//############################################################################
// Local time; used for timestamps
//############################################################################
GVL_MSG_XTS.fbLocalTime();
GVL_MSG_XTS.sLocalTime                              := GVL_MSG_XTS.fbLocalTime.LocalTimeString;
GVL_MSG_XTS.dtLocalTime                             := GVL_MSG_XTS.fbLocalTime.LocalTime;
//############################################################################
//############################################################################
// 	example for init sequence
//############################################################################	
CASE eInit
OF
  E_PROGRESS.PROGRESS_INVALID:
    // In the beginning there was no error...
    eInitError                                  := E_PROGRESS.PROGRESS_NOT_EXIST;
    //---------------------------------------------------------------------------
    // where are the stations?
    // TODO: after importing this project into your XTS TwinCAT solution
    //       setup of Station parameters is required.
    //---------------------------------------------------------------------------
    // default initialization, please leave this in here
    DefaultStationParameters();        
    //---------------------------------------------------------------------------
    //---------------------------------------------------------------------------
    // where to start?
    // fb_TransportUnit is connected StationStartIndex and StationStart
    //
    // TODO: after importing this project into your XTS TwinCAT solution
    //       setup of StartStation parameters is up to you to decide.
    //---------------------------------------------------------------------------
    GVL_XTS.StationStartIndex                   := 1; // this index is yours to change, fbTransportUnit is connected to it
    GVL_XTS.StationStart                        := GVL_XTS.StationParameter[GVL_XTS.StationStartIndex]; // put in here any plausible data you like
    //---------------------------------------------------------------------------

    eInit                                       := E_PROGRESS.PROGRESS_BUSY;
    // clear command interface
    GVL_XTS.XpuCtrl.Cmd                         := E_XPU_CTRL.XTS_CMD_NULL;
    GVL_MSG_XTS.TransportMessageCtrl.Cmd            := E_MESSAGE_CTRL.MSG_CTRL_NULL;
    GVL_MSG_XTS.MetricsMessageCtrl.Cmd              := E_MESSAGE_CTRL.MSG_CTRL_NULL;

    // set detailed message levvel for startup
    GVL_MSG_XTS.MessageLevelXpu                     := E_MessageType.eMessageVerbose; //GVL_MSG.MessageLevel;
    GVL_XTS.CaGroup.MessageLevel                := E_MessageType.eMessageVerbose; //GVL_MSG.MessageLevel;
    GVL_XTS.XtsTransport.MessageLevel           := E_MessageType.eMessageVerbose; //GVL_MSG.MessageLevel;

    FOR nStation := 1 TO MAX_STATION
    DO
      GVL_MSG_XTS.MessageLevelStations[nStation]    := E_MessageType.eMessageVerbose; //GVL_MSG.MessageLevel;
    END_FOR
    FOR nMover := 1 TO MAX_MOVER
    DO
      GVL_MSG_XTS.MessageLevelMovers[nMover]        := E_MessageType.eMessageVerbose; //GVL_MSG.MessageLevel;
    END_FOR
    
  //-----------------------------------------------------------------------------
  //-----------------------------------------------------------------------------
  E_PROGRESS.PROGRESS_BUSY:         // init Xpu, ProcessingUnit, MotorModules
    eInit                                       := E_PROGRESS.PROGRESS_PREPARE;
    GVL_MSG_XTS.TransportMessageCtrl.Cmd            := E_MESSAGE_CTRL.MSG_CTRL_INIT;
    GVL_MSG_XTS.MetricsMessageCtrl.Cmd              := E_MESSAGE_CTRL.MSG_CTRL_INIT;


  //-----------------------------------------------------------------------------
  //-----------------------------------------------------------------------------
  E_PROGRESS.PROGRESS_PREPARE:      // wait for init to be done
    GVL_XTS.XpuCtrl.Cmd                         := E_XPU_CTRL.XTS_CMD_INIT;
    IF (GVL_XTS.XpuState.State      = E_XPU_STATE.XTS_INIT + E_PROGRESS.PROGRESS_ERROR)
    THEN
      stMsg.eType                               := E_MessageType.eMessageInfo;
      stMsg.eDevice                             := e_Device.Device_Main;
      stMsg.eSubdevice                          := e_Subdevice.MainInit;
      stMsg.iErrorNumber                        := GVL_XTS.XpuState.Check;
      stMsg.sText                               := concat('MAIN.eInit Error: ', TO_STRING(MAIN_XTS.eInit));
      stMsg.sText                               := concat(stMsg.sText , ': ');
      stMsg.sText                               := concat(stMsg.sText, 'XpuState.Check: ');
      stMsg.sText                               := concat(stMsg.sText, TO_STRING(GVL_XTS.XpuState.Check));
      f_MessageSet(stMsg);

      eInitError                                := eInit;
      eInit                                     := E_PROGRESS.PROGRESS_ERROR;

    ELSIF (GVL_XTS.XpuState.State   = E_XPU_STATE.XTS_INIT + E_PROGRESS.PROGRESS_DONE)
    THEN
      eInit                                     := E_PROGRESS.PROGRESS_STARTUP;
      GVL_XTS.XpuCtrl.Cmd                       := E_XPU_CTRL.XTS_IDLE;
    END_IF

  //-----------------------------------------------------------------------------
  //-----------------------------------------------------------------------------
  E_PROGRESS.PROGRESS_STARTUP:
    CASE GVL_XTS.XpuState.Check
    OF
      E_XPU_CHECK.MOVER_ID_SIMULATION,
      E_XPU_CHECK.MOVER_ID_DETECTION_VALID:
        IF (GVL_XTS.XpuState.State = E_XPU_STATE.XTS_IDLE + E_PROGRESS.PROGRESS_WORKING)
        THEN
          eInit                                     := E_PROGRESS.PROGRESS_CHECK;
        END_IF
    END_CASE
  //-----------------------------------------------------------------------------
  //-----------------------------------------------------------------------------
  E_PROGRESS.PROGRESS_CHECK:
    eInit                                       := E_PROGRESS.PROGRESS_OCCUPIED;

    FOR nStation := 1 TO MAX_STATION
    DO
      GVL_MSG_XTS.MessageLevelStations[nStation]    := GVL_MSG_XTS.MessageLevel;
    END_FOR
    FOR nMover := 1 TO MAX_MOVER
    DO
      GVL_MSG_XTS.MessageLevelMovers[nMover]        := GVL_MSG_XTS.MessageLevel;
    END_FOR

  //-----------------------------------------------------------------------------
  //-----------------------------------------------------------------------------
  E_PROGRESS.PROGRESS_OCCUPIED:
    //---------------------------------------------------------------------------
    // how many nests to start with?
    // - this is for you to decide and me to secure, 
    //    so leave the initialisation as it is
    //
    // TODO: after importing this project into your XTS TwinCAT solution
    //       setup of StartStation NestMask configuration is up to you to decide.
    //---------------------------------------------------------------------------
    IF (GVL_XTS.XtsTransport.StationStartIndex > 0) AND
       (GVL_XTS.XtsTransport.StationStartIndex < MAX_STATION+1)
    THEN
      GVL_XTS.StationStart.nConfiguredStopCount := GVL_XTS.StationParameter[GVL_XTS.XtsTransport.StationStartIndex].nConfiguredStopCount;
    END_IF
    eInit                                       := E_PROGRESS.PROGRESS_WORKING;

  //-----------------------------------------------------------------------------
  //-----------------------------------------------------------------------------
  E_PROGRESS.PROGRESS_WORKING:
    GVL_MSG_XTS.TransportMessageCtrl.Cmd            := E_MESSAGE_CTRL.MSG_CTRL_WRITE;
    eInit                                       := E_PROGRESS.PROGRESS_DONE;

    stMsg.eType                                 := E_MessageType.eMessageInfo;
    stMsg.eDevice                               := e_Device.Device_Main;
    stMsg.eSubdevice                            := e_Subdevice.MainInit;
    stMsg.iErrorNumber                          := GVL_XTS.XpuState.Check;
    stMsg.sText                                 := concat('MAIN.eInit Done: ', TO_STRING(MAIN_XTS.eInit));
    stMsg.sText                                 := concat(stMsg.sText , ': ');
    stMsg.sText                                 := concat(stMsg.sText, 'XpuState.Check: ');
    stMsg.sText                                 := concat(stMsg.sText, TO_STRING(GVL_XTS.XpuState.Check));
    f_MessageSet(stMsg);

    //---------------------------------------------------------------------------
END_CASE
//############################################################################
//############################################################################
// 	/XTS Transport Unit
//############################################################################
//  - main control function block for transport layer
//  - requires access to member controls
//    - Xpu
//    - CaGroup
//    - Mover
//    - Station Control
//    - Station LinkedList Interface
//############################################################################
//
// cyclic call
GVL_XTS.XtsTransport();

// main control
GVL_XTS.XtsTransport.Ctrl                       REF= GVL_XTS.XtsTransportCtrl;   // main control
GVL_XTS.XtsTransport.State                      REF= GVL_XTS.XtsTransportState;  // main state
                                        
// member controls                      
GVL_XTS.XtsTransport.XpuCtrl                    REF= GVL_XTS.XpuCtrl;
GVL_XTS.XtsTransport.XpuState                   REF= GVL_XTS.XpuState;
GVL_XTS.XtsTransport.XpuInfo                    REF= GVL_XTS.XpuInfo;
                                        
GVL_XTS.XtsTransport.GroupItf                   :=   GVL_XTS.CaGroupItf;
GVL_XTS.XtsTransport.GroupInfo                  REF= GVL_XTS.CaGroupInfo;
                                        
GVL_XTS.XtsTransport.MoverItf                   REF= GVL_XTS.MoverItf;
GVL_XTS.XtsTransport.MoverInfo                  REF= GVL_XTS.MoverInfo;
GVL_XTS.XtsTransport.MoverLastPosition          REF= GVL_XTS.LastPosition;
GVL_XTS.XtsTransport.MoverLastGap               REF= GVL_XTS.LastGap;

GVL_XTS.XtsTransport.StationStartIndex          :=   GVL_XTS.StationStartIndex;                                        
GVL_XTS.XtsTransport.StationStart               REF= GVL_XTS.StationStart;      // start position for E_XTS_TRANSPORT_CTRL.CMD_TRANSPORT_START
GVL_XTS.XtsTransport.StationCtrlItf             REF= GVL_XTS.StationCtrlItf;    // station interfaces are required for accessing station methods
GVL_XTS.XtsTransport.StationListsItf            REF= GVL_XTS.StationListItf;    // list interface is required for access to linked list methods
GVL_XTS.XtsTransport.StationControl             REF= GVL_XTS.StationCtrl;
GVL_XTS.XtsTransport.StationState               REF= GVL_XTS.StationState;
//############################################################################
// 	XTS Transport Unit/
//############################################################################
//############################################################################
//############################################################################
// 	/XTS Stations
//############################################################################	
FOR nStation := 1 TO MAX_STATION
DO
  // epimetheus assembles the body
  GVL_XTS.StationListItf[nStation]              := GVL_XTS.StationList[nStation];   // interfaces for list methods
  GVL_XTS.StationCtrlItf[nStation]              := GVL_XTS.Station[nStation];       // interfaces for station methods

  CASE GVL_XTS.StationParameter[nStation].eType
  OF
    //-----------------------------------------------------------------------------
    E_STATION_TYPE.STATION_PROCESS:
      GVL_XTS.Station[nStation].MessageLevel    := GVL_MSG_XTS.MessageLevelStations[nStation];

      GVL_XTS.Station[nStation].StationId       := nStation;  // Know Thyself!

    
      GVL_XTS.Station[nStation].Ctrl            REF= GVL_XTS.StationCtrl;           // station ctrl from extern
      GVL_XTS.Station[nStation].State           REF= GVL_XTS.StationState;          // station state to extern
    
      GVL_XTS.Station[nStation].ItfStations     REF= GVL_XTS.StationListItf;        // give every station all list interfaces for writing mover tickets
      GVL_XTS.Station[nStation].ItfMover        REF= GVL_XTS.MoverItf;              // give every station all mover interfaces for movement in / out of station
      GVL_XTS.Station[nStation].Mover           REF= GVL_XTS.AxisRefMover;          // AXIS_REF to read infos from
      GVL_XTS.Station[nStation].MoverOffset     REF= GVL_XTS.PositionOffset;        // static offsets for all stations, all movers, all stop positions
    
      GVL_XTS.Station[nStation].StationParameter  REF= GVL_XTS.StationParameter;// give every station all station parameters for sending to WaitPos of target station
    
      // cyclic call
      GVL_XTS.Station[nStation].Cycle();                                        // cycle for handshaking with extern
    
      // Queue data for each station
      GVL_XTS.StationQueue[nStation]            := GVL_XTS.StationListItf[nStation].Data;


    //-----------------------------------------------------------------------------
    E_STATION_TYPE.STATION_GEAR_IN_POS:
      GVL_XTS.StationGearIn[nStation].MessageLevel:= GVL_MSG_XTS.MessageLevelStations[nStation];

      GVL_XTS.StationGearIn[nStation].StationId   := nStation;  // Know Thyself!
    
      GVL_XTS.StationGearIn[nStation].Ctrl        REF= GVL_XTS.StationCtrl;           // station ctrl from extern
      GVL_XTS.StationGearIn[nStation].State       REF= GVL_XTS.StationState;          // station state to extern
    
      GVL_XTS.StationGearIn[nStation].ItfStations REF= GVL_XTS.StationListItf;        // give every station all list interfaces for writing mover tickets
      GVL_XTS.StationGearIn[nStation].ItfMover    REF= GVL_XTS.MoverItf;              // give every station all mover interfaces for movement in / out of station
      GVL_XTS.StationGearIn[nStation].Mover       REF= GVL_XTS.AxisRefMover;          // AXIS_REF to read infos from
      GVL_XTS.StationGearIn[nStation].MoverOffset REF= GVL_XTS.PositionOffset;        // static offsets for all stations, all movers, all stop positions
    
    
      GVL_XTS.StationGearIn[nStation].StationParameter  REF= GVL_XTS.StationParameter;// give every station all station parameters for sending to WaitPos of target station
    
      // cyclic call
      GVL_XTS.StationGearIn[nStation].Cycle();                                        // cycle for handshaking with extern
    
      // Queue data for each station
      GVL_XTS.StationQueue[nStation]            := GVL_XTS.StationListItf[nStation].Data;
  ELSE
      //---------------------------------------------------------------------------------
      // no valid station type --> no identity
      //---------------------------------------------------------------------------------
      GVL_XTS.Station[nStation].StationId       := 0; // I am no one
      //---------------------------------------------------------------------------------
  END_CASE
END_FOR
//############################################################################
// 	XTS Stations/
//############################################################################	
//############################################################################
//############################################################################
// 	/XPU environment
//############################################################################	
GVL_XTS.Xpu.XpuInstance                         :=   1;
GVL_XTS.Xpu.MessageLevel                        :=   GVL_MSG_XTS.MessageLevelXpu;

GVL_XTS.Xpu.Ctrl                                REF= GVL_XTS.XpuCtrl;
GVL_XTS.Xpu.State                               REF= GVL_XTS.XpuState;
GVL_XTS.Xpu.XpuModuleInfoData                   REF= GVL_XTS.XpuModules;

GVL_XTS.Xpu.CaGroupOID                          :=   GVL_XTS.CaGroup.GroupInfo.CaGroupOID;

// cyclic call                                
GVL_XTS.Xpu();                                
GVL_XTS.XpuInfo                                 :=   GVL_XTS.Xpu.XpuInfo;
//############################################################################
// 	XPU environment/
//############################################################################	
//############################################################################
//############################################################################	
// 	/CA-Group Class
//############################################################################
// message device identifier
GVL_XTS.CaGroup.MessageDeviceIndex              :=   e_Device.CaGroup + 1;	
// assignment
GVL_XTS.CaGroup.AxisRef                         REF= GVL_XTS.AxisRefMover;
// Interface to Mover methods
GVL_XTS.CaGroup.MoverItf                        REF= GVL_XTS.MoverItf; 
GVL_XTS.CaGroup.GroupRef                        REF= GVL_XTS.CaGroupRef;
GVL_XTS.CaGroup.XpuInfo                         REF= GVL_XTS.XpuInfo;
// cyclic call
GVL_XTS.CaGroup.InfoCycle(TRUE);                // read group status
// InfoData from group
GVL_XTS.CaGroupInfo                             :=   GVL_XTS.CaGroup.GroupInfo;
// Interface of CaGroup
GVL_XTS.CaGroupItf                              :=   GVL_XTS.CaGroup;
//############################################################################	
// 	CA-Group Class/
//############################################################################
//############################################################################
//############################################################################
//  /Mover Class	
//############################################################################	
FOR nMover := 1 TO MAX_MOVER
DO
  GVL_XTS.Mover[nMover].MoverId                 :=   nMover;
  GVL_XTS.Mover[nMover].RailLength              :=   GVL_XTS.Xpu.RailLength;  // mover needs RailLength, in order to calc absolute position from modulo input
  GVL_XTS.Mover[nMover].MessageLevel            :=   GVL_MSG_XTS.MessageLevelMovers[nMover];

  GVL_XTS.Mover[nMover].Ctrl                    REF= GVL_XTS.MoverCtrl;       // mover control from extern
  GVL_XTS.Mover[nMover].State                   REF= GVL_XTS.MoverState;      // mover state to extern

  GVL_XTS.Mover[nMover].MoveData                REF= GVL_XTS.MoveData;        // dyn constraints for extern to write
  GVL_XTS.Mover[nMover].GearData                REF= GVL_XTS.GearData;        // GearIn/GearInPosCa data fro extern to write

  // assignment
  GVL_XTS.Mover[nMover].Mover                   REF= GVL_XTS.AxisRefMover[nMover];  // axis reference to Mover function block
  GVL_XTS.Mover[nMover].LastGap                 REF= GVL_XTS.LastGap[nMover];       // reference to last used gap value datafield
  GVL_XTS.Mover[nMover].LastPosition            REF= GVL_XTS.LastPosition[nMover];  // reference to last position datafield

  GVL_XTS.Mover[nMover].MoverInfo		            REF= GVL_XTS.MoverInfo[nMover];     // refernence to mover info data (ActPos, SetPos, ...)

  GVL_XTS.MoverItf[nMover]                      :=   GVL_XTS.Mover[nMover];

  // cyclic call
  GVL_XTS.Mover[nMover].Cycle();                // call AXIS_REF()
  GVL_XTS.Mover[nMover]();                      // call Ctrl/State
END_FOR
//############################################################################
//  Mover Class/	
//############################################################################	
//############################################################################
//############################################################################
//  /Mover Selector	
//############################################################################
GVL_XTS.MoverSelector.Ctrl                      REF= GVL_XTS.MoverSelectorCtrl;
GVL_XTS.MoverSelector.State                     REF= GVL_XTS.MoverSelectorState;
GVL_XTS.MoverSelector.AxisRef                   REF= GVL_XTS.AxisRefMover;
GVL_XTS.MoverSelector.Info                      REF= GVL_XTS.MoverInfo;
GVL_XTS.MoverSelector.ItfMover                  REF= GVL_XTS.MoverItf;

GVL_XTS.MoverSelector();
//############################################################################
//  Mover Selector/	
//############################################################################	
//############################################################################
//############################################################################
//  /logging
//    - all life is problem solving
//############################################################################
GVL_MSG_XTS.TransportMessageData.Ctrl               REF= GVL_MSG_XTS.TransportMessageCtrl;
GVL_MSG_XTS.TransportMessageData.State              REF= GVL_MSG_XTS.TransportMessageState;
GVL_MSG_XTS.TransportMessageData.MessageIndex       REF= GVL_MSG_XTS.MessageTransportIndex;
GVL_MSG_XTS.TransportMessageData.ErrorIndex         REF= GVL_MSG_XTS.MessageTransportError;
GVL_MSG_XTS.TransportMessageData.DirRoot            :=   ADR(GVL_MSG_XTS.LOG_DIR);
GVL_MSG_XTS.TransportMessageData.FileRoot           :=   ADR(GVL_MSG_XTS.LOG_FILE);
GVL_MSG_XTS.TransportMessageData.MsgList            :=   ADR(GVL_MSG_XTS.TransportMessages);
GVL_MSG_XTS.TransportMessageData.LocalTime          :=   ADR(GVL_MSG_XTS.dtLocalTime);
GVL_MSG_XTS.TransportMessageData();
eMsgState                                       :=   f_GetState   (GVL_MSG_XTS.TransportMessageState.State);
eMsgProgress                                    :=   f_GetProgress(GVL_MSG_XTS.TransportMessageState.State);

CASE eMsgState
OF
  E_MESSAGE_STATE.MSG_STATE_NULL:
    CASE eMsgProgress
    OF
      E_PROGRESS.PROGRESS_INVALID,
      E_PROGRESS.PROGRESS_DONE:
        IF (GVL_MSG_XTS.MessageTransportIndex > GVL_MSG_XTS.MAX_MESSAGE/100) OR
           (GVL_MSG_XTS.MessageTransportError > 0)
        THEN
          GVL_MSG_XTS.TransportMessageCtrl.Cmd      := E_MESSAGE_CTRL.MSG_CTRL_WRITE;
        ELSE
          tonIdleWriteMotion(IN := TRUE, PT:= tIdleWriteMotion);
          IF (tonIdleWriteMotion.Q)
          THEN
            GVL_MSG_XTS.TransportMessageCtrl.Cmd    := E_MESSAGE_CTRL.MSG_CTRL_WRITE;
          END_IF
        END_IF
    END_CASE

  E_MESSAGE_STATE.MSG_STATE_WRITE:
    CASE eMsgProgress
    OF
      E_PROGRESS.PROGRESS_ERROR,
      E_PROGRESS.PROGRESS_DONE:
          tonIdleWriteMotion(IN := FALSE, PT:= tIdleWriteMotion);
        GVL_MSG_XTS.TransportMessageCtrl.Cmd        := E_MESSAGE_CTRL.MSG_CTRL_NULL;
    END_CASE

ELSE
    CASE eMsgProgress
    OF
      E_PROGRESS.PROGRESS_DONE:
        GVL_MSG_XTS.TransportMessageCtrl.Cmd        := E_MESSAGE_CTRL.MSG_CTRL_NULL;
    END_CASE
END_CASE
//############################################################################
//  logging/
//############################################################################
//############################################################################
//############################################################################
//  /Transport Metrics
//############################################################################
GVL_MSG_XTS.MetricsMessageData.Ctrl                 REF= GVL_MSG_XTS.MetricsMessageCtrl;
GVL_MSG_XTS.MetricsMessageData.State                REF= GVL_MSG_XTS.MetricsMessageState;

GVL_MSG_XTS.MetricsMessageData.MessageIndex         REF= GVL_MSG_XTS.MessageMetricsIndex;
GVL_MSG_XTS.MetricsMessageData.ErrorIndex           REF= GVL_MSG_XTS.MessageMetricsError;

GVL_MSG_XTS.MetricsMessageData.DirRoot              :=   ADR(GVL_MSG_XTS.LOG_DIR);
GVL_MSG_XTS.MetricsMessageData.FileRoot             :=   ADR(GVL_MSG_XTS.LOG_FILE_METRIC);

GVL_MSG_XTS.MetricsMessageData.MsgList              :=   ADR(GVL_MSG_XTS.MetricsMessages);
GVL_MSG_XTS.MetricsMessageData.LocalTime            :=   ADR(GVL_MSG_XTS.dtLocalTime);

GVL_MSG_XTS.MetricsMessageData();

eMtrState                                       := f_GetState   (GVL_MSG_XTS.MetricsMessageState.State);
eMtrProgress                                    := f_GetProgress(GVL_MSG_XTS.MetricsMessageState.State);

CASE eMtrState
OF
  E_MESSAGE_STATE.MSG_STATE_NULL:
    CASE eMtrProgress
    OF
      E_PROGRESS.PROGRESS_INVALID:
        IF (GVL_MSG_XTS.MessageMetricsIndex > GVL_MSG_XTS.MAX_MESSAGE/100) OR
           (GVL_MSG_XTS.MessageMetricsError > 0)
        THEN
          GVL_MSG_XTS.MetricsMessageCtrl.Cmd        := E_MESSAGE_CTRL.MSG_CTRL_WRITE;
        ELSE
          tonIdleWriteMetric(IN := TRUE, PT:= tIdleWriteMetric);
          IF (tonIdleWriteMetric.Q)
          THEN
            GVL_MSG_XTS.MetricsMessageCtrl.Cmd      := E_MESSAGE_CTRL.MSG_CTRL_WRITE;
          END_IF
        END_IF
    END_CASE

  E_MESSAGE_STATE.MSG_STATE_WRITE:
    CASE eMtrProgress
    OF
      E_PROGRESS.PROGRESS_ERROR,
      E_PROGRESS.PROGRESS_DONE:
        tonIdleWriteMetric(IN := FALSE, PT:= tIdleWriteMetric);
        GVL_MSG_XTS.MetricsMessageCtrl.Cmd          := E_MESSAGE_CTRL.MSG_CTRL_NULL;
    END_CASE
ELSE
    CASE eMtrProgress
    OF
      E_PROGRESS.PROGRESS_DONE:
        GVL_MSG_XTS.MetricsMessageCtrl.Cmd          := E_MESSAGE_CTRL.MSG_CTRL_NULL;
    END_CASE
END_CASE
//############################################################################
//  Transport Metrics/
//############################################################################
//############################################################################
//############################################################################
//  /Visualization data	
//############################################################################
VisualizationData();
//############################################################################
//  Visualization data/	
//############################################################################

ACTION DefaultStationParameters:
//---------------------------------------------------------------------------------------
//---------------------------------------------------------------------------------------
//
//  Default Station dynamics 
//  - we do not want an array full of nothing 
//  - better have something
//  - leave this initialisation as it is, 
//  - go to MAIN_APP to configure the global datafields
//
//---------------------------------------------------------------------------------------
//---------------------------------------------------------------------------------------
FOR nStn := 1 TO MAX_STATION
DO
  GVL_XTS.StationParameter[nStn].eType               :=   E_STATION_TYPE.INVALID; // make it valid in your configuration
  GVL_XTS.StationParameter[nStn].sText               :=   concat('DEaF_STATION_', TO_STRING(nStn));

  GVL_XTS.StationParameter[nStn].rPosWait            :=   TO_REAL(ABS(GVL_XTS.XpuInfo.rRailLength - nStn*10.0));
  GVL_XTS.StationParameter[nStn].rGap                :=   rInitGap;
  GVL_XTS.StationParameter[nStn].rVelo               :=   rInitVelo;
  GVL_XTS.StationParameter[nStn].rAccDec             :=   rInitAcc;
  GVL_XTS.StationParameter[nStn].rJerk               :=   rInitJerk;
END_FOR
//---------------------------------------------------------------------------------------
//---------------------------------------------------------------------------------------
END_ACTION

ACTION VisualizationData:
//############################################################################
//############################################################################
// Visualization data	
//############################################################################
// get enumerations from XPU for visu:	
eTransportState                       := f_GetState   (GVL_XTS.XtsTransportState.State);
eTransportResult                      := f_GetProgress(GVL_XTS.XtsTransportState.State);

eXpuState                             := f_GetState   (GVL_XTS.XtsTransportState.XpuState.State);
eXpuResult                            := f_GetProgress(GVL_XTS.XtsTransportState.XpuState.State);

eXpuCheck                             := GVL_XTS.XtsTransportState.XpuState.Check;

// display xpu state and result in visu
// get strings and info
sCaGroupState                         := TO_STRING(GVL_XTS.XtsTransportState.GroupInfo.CaGroupState);

sTransportState                       := TO_STRING(eTransportState);
sTransportCheck                       := TO_STRING(GVL_XTS.XtsTransportState.Check);
sTransportResult                      := TO_STRING(eTransportResult);

stXpuStrings.sXpuState                := TO_STRING(eXpuState);
stXpuStrings.sXpuResult               := TO_STRING(eXpuResult);
stXpuStrings.sXpuCyclicCheck          := TO_STRING(eXpuCheck);

stXpuStrings.sXpuOpMode               := GVL_XTS.Xpu.OpModeToString();
stXpuStrings.sXpuMoverId_DetectionMode:= GVL_XTS.Xpu.IdDetectionModeToString();
stXpuStrings.sXpuMoverPosAssignement  := GVL_XTS.Xpu.MoverPositionAssignementToString();

nMoverSelected                        := SEL((nMoverSelected<1), nMoverSelected, 1);
nMoverSelected                        := SEL((nMoverSelected>MAX_MOVER), nMoverSelected, MAX_MOVER);

nStationSelected                      := SEL((nStationSelected<1), nStationSelected, 1);
nStationSelected                      := SEL((nStationSelected>MAX_STATION), nStationSelected, MAX_STATION);

bStationEnable                        := SEL((GVL_XTS.StationCtrl[nStationSelected].Cmd = E_STATION_CTRL.STATION_ENABLE),        FALSE, TRUE);
bStationEnter                         := SEL((GVL_XTS.StationCtrl[nStationSelected].Cmd = E_STATION_CTRL.STATION_MOVER_ENTER),   FALSE, TRUE);
bStationStart                         := SEL((GVL_XTS.StationCtrl[nStationSelected].Cmd = E_STATION_CTRL.STATION_PROCESS_START), FALSE, TRUE);
bStationDone                          := SEL((GVL_XTS.StationCtrl[nStationSelected].Cmd = E_STATION_CTRL.STATION_PROCESS_DONE),  FALSE, TRUE);
bStationOut                           := SEL((GVL_XTS.StationCtrl[nStationSelected].Cmd = E_STATION_CTRL.STATION_MOVER_OUT),     FALSE, TRUE);
bStationGone                          := SEL((GVL_XTS.StationCtrl[nStationSelected].Cmd = E_STATION_CTRL.STATION_MOVER_GONE),    FALSE, TRUE);

eMoverState                           := f_GetState   (GVL_XTS.MoverState[nMoverSelected].State);
eMoverResult                          := f_GetProgress(GVL_XTS.MoverState[nMoverSelected].State);

sMoverState                           := TO_STRING(eMoverState);
sMoverResult                          := TO_STRING(eMoverResult);

eSelectorState                        := f_GetState   (GVL_XTS.MoverSelectorState.State.State);
eSelectorResult                       := f_GetProgress(GVL_XTS.MoverSelectorState.State.State);

sSelectorState                        := TO_STRING(eSelectorState);
sSelectorResult                       := TO_STRING(eSelectorResult);

sStationState                         := TO_STRING(GVL_XTS.StationState[nStationSelected].State);
sStationStateMask                     := Tc2_Utilities.BYTE_TO_BINSTR(GVL_XTS.StationState[nStationSelected].nMask, 8);
sStationCtrlMask                      := Tc2_Utilities.BYTE_TO_BINSTR(GVL_XTS.StationCtrl[nStationSelected].nMask, 8);

tStationSelectedQueue                 := GVL_XTS.StationQueue[nStationSelected];
//############################################################################
//############################################################################
END_ACTION

END_PROGRAM

// ---- APPLICATION/StationPrimesExample.TcPOU
FUNCTION StationPrimesExample : bool
VAR
  nStationParameter           : UINT;
END_VAR

//-----------------------------------------------------------------------------------------------------------------------------------------
//-----------------------------------------------------------------------------------------------------------------------------------------
//
//  HAUD 2026.04.30
//
//  - StationPrimes example
//
//  - hard coded station parameters as example
//  - TODO: xml DataServer implementation for station parameter read/write
//
//  - reminder: (this you HAVE to check manually when setting up the transport)
//-----------------------------------------------------------------------------
//    - DO NOT place the modulo turn within the range of a station
//
//    - in case the extern process requires multiple xts stations, 
//      - the range must be closed and in strict order
//-----------------------------------------------------------------------------------------------------------------------------------------
//-----------------------------------------------------------------------------------------------------------------------------------------
//-----------------------------------------------------------------------------------------------------------------------------------------
// THIS IS ONLY FOR EXAMPLE USE, 
//  CHECK GVL_XTS.MAX_STATION MANUALLY
//-----------------------------------------------------------------------------------------------------------------------------------------
//---------------------------------------------------------------------------------------
//---------------------------------------------------------------------------------------
nStationParameter                    := 1;
GVL_XTS.StationParameter[nStationParameter].eType               := E_STATION_TYPE.STATION_PROCESS;
GVL_XTS.StationParameter[nStationParameter].sText               := 'ST011';
GVL_XTS.StationParameter[nStationParameter].rPosWait            :=     10.0; // absolute modulo position
GVL_XTS.StationParameter[nStationParameter].rPosStop[1]         :=     90.0; // relative to rPosWait
GVL_XTS.StationParameter[nStationParameter].rReleaseDistance    :=     80.0; // relative to Mover.ActPos
GVL_XTS.StationParameter[nStationParameter].rVelo               :=   2500.0;

nStationParameter                    := 2;
GVL_XTS.StationParameter[nStationParameter].eType               := E_STATION_TYPE.STATION_PROCESS;
GVL_XTS.StationParameter[nStationParameter].sText               := 'ST012';
GVL_XTS.StationParameter[nStationParameter].rPosWait            :=     10.0; // absolute modulo position
GVL_XTS.StationParameter[nStationParameter].rPosStop[1]         :=    180.0; // relative to rPosWait
GVL_XTS.StationParameter[nStationParameter].rReleaseDistance    :=     40.0; // relative to Mover.ActPos
GVL_XTS.StationParameter[nStationParameter].rVelo               :=   2500.0;

nStationParameter                    := 3;
GVL_XTS.StationParameter[nStationParameter].eType               := E_STATION_TYPE.STATION_PROCESS;
GVL_XTS.StationParameter[nStationParameter].sText               := 'ST013';
GVL_XTS.StationParameter[nStationParameter].rPosWait            :=     10.0; // absolute modulo position
GVL_XTS.StationParameter[nStationParameter].rPosStop[1]         :=    270.0; // relative to rPosWait
GVL_XTS.StationParameter[nStationParameter].rReleaseDistance    :=     10.0; // relative to Mover.ActPos
GVL_XTS.StationParameter[nStationParameter].rVelo               :=   2500.0;

//---------------------------------------------------------------------------------------
//---------------------------------------------------------------------------------------
nStationParameter                    := 4;
GVL_XTS.StationParameter[nStationParameter].eType               := E_STATION_TYPE.STATION_PROCESS;
GVL_XTS.StationParameter[nStationParameter].sText               := 'ST021';
GVL_XTS.StationParameter[nStationParameter].rPosWait            :=    600.0; // absolute modulo position
GVL_XTS.StationParameter[nStationParameter].rPosStop[1]         :=      0.0; // relative to rPosWait
GVL_XTS.StationParameter[nStationParameter].rReleaseDistance    :=     70.0; // relative to Mover.ActPos
GVL_XTS.StationParameter[nStationParameter].rVelo               :=   2500.0;

nStationParameter                    := 5;
GVL_XTS.StationParameter[nStationParameter].eType               := E_STATION_TYPE.STATION_PROCESS;
GVL_XTS.StationParameter[nStationParameter].sText               := 'ST022';
GVL_XTS.StationParameter[nStationParameter].rPosWait            :=    690.0; // absolute modulo position
GVL_XTS.StationParameter[nStationParameter].rPosStop[1]         :=      0.0; // relative to rPosWait
GVL_XTS.StationParameter[nStationParameter].rReleaseDistance    :=     45.0; // relative to Mover.ActPos
GVL_XTS.StationParameter[nStationParameter].rVelo               :=   2500.0;

nStationParameter                    := 6;
GVL_XTS.StationParameter[nStationParameter].eType               := E_STATION_TYPE.STATION_PROCESS;
GVL_XTS.StationParameter[nStationParameter].sText               := 'ST023';
GVL_XTS.StationParameter[nStationParameter].rPosWait            :=    780.0; // absolute modulo position
GVL_XTS.StationParameter[nStationParameter].rPosStop[1]         :=      0.0; // relative to rPosWait
GVL_XTS.StationParameter[nStationParameter].rReleaseDistance    :=     25.0; // relative to Mover.ActPos
GVL_XTS.StationParameter[nStationParameter].rVelo               :=   2500.0;


nStationParameter                    := 7;
GVL_XTS.StationParameter[nStationParameter].eType               := E_STATION_TYPE.STATION_PROCESS;
GVL_XTS.StationParameter[nStationParameter].sText               := 'ST024';
GVL_XTS.StationParameter[nStationParameter].rPosWait            :=    870.0; // absolute modulo position
GVL_XTS.StationParameter[nStationParameter].rPosStop[1]         :=      0.0; // relative to rPosWait
GVL_XTS.StationParameter[nStationParameter].rReleaseDistance    :=     10.0; // relative to Mover.ActPos
GVL_XTS.StationParameter[nStationParameter].rVelo               :=   2500.0;

//---------------------------------------------------------------------------------------
//---------------------------------------------------------------------------------------
nStationParameter                    := 8;
GVL_XTS.StationParameter[nStationParameter].eType               := E_STATION_TYPE.STATION_PROCESS;
GVL_XTS.StationParameter[nStationParameter].sText               := 'ST031';
GVL_XTS.StationParameter[nStationParameter].rPosWait            :=   1500.0; // absolute modulo position
GVL_XTS.StationParameter[nStationParameter].rPosStop[1]         :=     90.0; // relative to rPosWait
GVL_XTS.StationParameter[nStationParameter].rReleaseDistance    :=    110.0; // relative to Mover.ActPos
GVL_XTS.StationParameter[nStationParameter].rVelo               :=   2500.0;

nStationParameter                    := 9;
GVL_XTS.StationParameter[nStationParameter].eType               := E_STATION_TYPE.STATION_PROCESS;
GVL_XTS.StationParameter[nStationParameter].sText               := 'ST032';
GVL_XTS.StationParameter[nStationParameter].rPosWait            :=   1500.0; // absolute modulo position
GVL_XTS.StationParameter[nStationParameter].rPosStop[1]         :=    180.0; // relative to rPosWait
GVL_XTS.StationParameter[nStationParameter].rReleaseDistance    :=     70.0; // relative to Mover.ActPos
GVL_XTS.StationParameter[nStationParameter].rVelo               :=   2500.0;

nStationParameter                    := 10;
GVL_XTS.StationParameter[nStationParameter].eType               := E_STATION_TYPE.STATION_PROCESS;
GVL_XTS.StationParameter[nStationParameter].sText               := 'ST033';
GVL_XTS.StationParameter[nStationParameter].rPosWait            :=   1500.0; // absolute modulo position
GVL_XTS.StationParameter[nStationParameter].rPosStop[1]         :=    270.0; // relative to rPosWait
GVL_XTS.StationParameter[nStationParameter].rReleaseDistance    :=     45.0; // relative to Mover.ActPos
GVL_XTS.StationParameter[nStationParameter].rVelo               :=   2500.0;

nStationParameter                    := 11;
GVL_XTS.StationParameter[nStationParameter].eType               := E_STATION_TYPE.STATION_PROCESS;
GVL_XTS.StationParameter[nStationParameter].sText               := 'ST034';
GVL_XTS.StationParameter[nStationParameter].rPosWait            :=   1500.0; // absolute modulo position
GVL_XTS.StationParameter[nStationParameter].rPosStop[1]         :=    360.0; // relative to rPosWait
GVL_XTS.StationParameter[nStationParameter].rReleaseDistance    :=     25.0; // relative to Mover.ActPos
GVL_XTS.StationParameter[nStationParameter].rVelo               :=   2500.0;

nStationParameter                    := 12;
GVL_XTS.StationParameter[nStationParameter].eType               := E_STATION_TYPE.STATION_PROCESS;
GVL_XTS.StationParameter[nStationParameter].sText               := 'ST035';
GVL_XTS.StationParameter[nStationParameter].rPosWait            :=   1500.0; // absolute modulo position
GVL_XTS.StationParameter[nStationParameter].rPosStop[1]         :=    450.0; // relative to rPosWait
GVL_XTS.StationParameter[nStationParameter].rReleaseDistance    :=     10.0; // relative to Mover.ActPos
GVL_XTS.StationParameter[nStationParameter].rVelo               :=   2500.0;

//---------------------------------------------------------------------------------------
//---------------------------------------------------------------------------------------
nStationParameter                    := 13;
GVL_XTS.StationParameter[nStationParameter].eType               := E_STATION_TYPE.STATION_PROCESS;
GVL_XTS.StationParameter[nStationParameter].sText               := 'ST041';
GVL_XTS.StationParameter[nStationParameter].rPosWait            :=   2900.0; // absolute modulo position
GVL_XTS.StationParameter[nStationParameter].rPosStop[1]         :=      0.0; // relative to rPosWait
GVL_XTS.StationParameter[nStationParameter].rPosStop[2]         :=     45.0; // relative to rPosWait
GVL_XTS.StationParameter[nStationParameter].rReleaseDistance    :=    500.0; // relative to Mover.ActPos
GVL_XTS.StationParameter[nStationParameter].rVelo               :=   2500.0;
GVL_XTS.StationParameter[nStationParameter].nConfiguredStopCount:= 2;

nStationParameter                    := 14;
GVL_XTS.StationParameter[nStationParameter].eType               := E_STATION_TYPE.STATION_PROCESS;
GVL_XTS.StationParameter[nStationParameter].sText               := 'ST042';
GVL_XTS.StationParameter[nStationParameter].rPosWait            :=   3000.0; // absolute modulo position
GVL_XTS.StationParameter[nStationParameter].rPosStop[1]         :=      0.0; // relative to rPosWait
GVL_XTS.StationParameter[nStationParameter].rPosStop[2]         :=     45.0; // relative to rPosWait
GVL_XTS.StationParameter[nStationParameter].rReleaseDistance    :=    400.0; // relative to Mover.ActPos
GVL_XTS.StationParameter[nStationParameter].rVelo               :=   2500.0;
GVL_XTS.StationParameter[nStationParameter].nConfiguredStopCount:= 2;

nStationParameter                    := 15;
GVL_XTS.StationParameter[nStationParameter].eType               := E_STATION_TYPE.STATION_PROCESS;
GVL_XTS.StationParameter[nStationParameter].sText               := 'ST043';
GVL_XTS.StationParameter[nStationParameter].rPosWait            :=   3100.0; // absolute modulo position
GVL_XTS.StationParameter[nStationParameter].rPosStop[1]         :=      0.0; // relative to rPosWait
GVL_XTS.StationParameter[nStationParameter].rPosStop[2]         :=     45.0; // relative to rPosWait
GVL_XTS.StationParameter[nStationParameter].rReleaseDistance    :=    300.0; // relative to Mover.ActPos
GVL_XTS.StationParameter[nStationParameter].rVelo               :=   2500.0;
GVL_XTS.StationParameter[nStationParameter].nConfiguredStopCount:= 2;

nStationParameter                    := 16;
GVL_XTS.StationParameter[nStationParameter].eType               := E_STATION_TYPE.STATION_PROCESS;
GVL_XTS.StationParameter[nStationParameter].sText               := 'ST044';
GVL_XTS.StationParameter[nStationParameter].rPosWait            :=   3200.0; // absolute modulo position
GVL_XTS.StationParameter[nStationParameter].rPosStop[1]         :=      0.0; // relative to rPosWait
GVL_XTS.StationParameter[nStationParameter].rPosStop[2]         :=     45.0; // relative to rPosWait
GVL_XTS.StationParameter[nStationParameter].rReleaseDistance    :=    200.0; // relative to Mover.ActPos
GVL_XTS.StationParameter[nStationParameter].rVelo               :=   2500.0;
GVL_XTS.StationParameter[nStationParameter].nConfiguredStopCount:= 2;

nStationParameter                    := 17;
GVL_XTS.StationParameter[nStationParameter].eType               := E_STATION_TYPE.STATION_PROCESS;
GVL_XTS.StationParameter[nStationParameter].sText               := 'ST045';
GVL_XTS.StationParameter[nStationParameter].rPosWait            :=   3300.0; // absolute modulo position
GVL_XTS.StationParameter[nStationParameter].rPosStop[1]         :=      0.0; // relative to rPosWait
GVL_XTS.StationParameter[nStationParameter].rPosStop[2]         :=     45.0; // relative to rPosWait
GVL_XTS.StationParameter[nStationParameter].rReleaseDistance    :=    100.0; // relative to Mover.ActPos
GVL_XTS.StationParameter[nStationParameter].rVelo               :=   2500.0;
GVL_XTS.StationParameter[nStationParameter].nConfiguredStopCount:= 2;

nStationParameter                    := 18;
GVL_XTS.StationParameter[nStationParameter].eType               := E_STATION_TYPE.STATION_PROCESS;
GVL_XTS.StationParameter[nStationParameter].sText               := 'ST046';
GVL_XTS.StationParameter[nStationParameter].rPosWait            :=   3400.0; // absolute modulo position
GVL_XTS.StationParameter[nStationParameter].rPosStop[1]         :=      0.0; // relative to rPosWait
GVL_XTS.StationParameter[nStationParameter].rPosStop[2]         :=     45.0; // relative to rPosWait
GVL_XTS.StationParameter[nStationParameter].rReleaseDistance    :=     10.0; // relative to Mover.ActPos
GVL_XTS.StationParameter[nStationParameter].rVelo               :=   2500.0;
GVL_XTS.StationParameter[nStationParameter].nConfiguredStopCount:= 2;

//---------------------------------------------------------------------------------------
//---------------------------------------------------------------------------------------
nStationParameter                    := 19;
GVL_XTS.StationParameter[nStationParameter].eType               := E_STATION_TYPE.STATION_PROCESS;
GVL_XTS.StationParameter[nStationParameter].sText               := 'ST051';
GVL_XTS.StationParameter[nStationParameter].rPosWait            :=   4100.0; // absolute modulo position
GVL_XTS.StationParameter[nStationParameter].rPosStop[1]         :=     90.0; // relative to rPosWait
GVL_XTS.StationParameter[nStationParameter].rPosStop[2]         :=    135.0; // relative to rPosWait
GVL_XTS.StationParameter[nStationParameter].rReleaseDistance    :=    200.0; // relative to Mover.ActPos
GVL_XTS.StationParameter[nStationParameter].rVelo               :=   2500.0;
GVL_XTS.StationParameter[nStationParameter].nConfiguredStopCount:= 2;

nStationParameter                    := 20;
GVL_XTS.StationParameter[nStationParameter].eType               := E_STATION_TYPE.STATION_PROCESS;
GVL_XTS.StationParameter[nStationParameter].sText               := 'ST052';
GVL_XTS.StationParameter[nStationParameter].rPosWait            :=   4100.0; // absolute modulo position
GVL_XTS.StationParameter[nStationParameter].rPosStop[1]         :=    180.0; // relative to rPosWait
GVL_XTS.StationParameter[nStationParameter].rPosStop[2]         :=    225.0; // relative to rPosWait
GVL_XTS.StationParameter[nStationParameter].rReleaseDistance    :=    100.0; // relative to Mover.ActPos
GVL_XTS.StationParameter[nStationParameter].rVelo               :=   2500.0;
GVL_XTS.StationParameter[nStationParameter].nConfiguredStopCount:= 2;

nStationParameter                    := 21;
GVL_XTS.StationParameter[nStationParameter].eType               := E_STATION_TYPE.STATION_PROCESS;
GVL_XTS.StationParameter[nStationParameter].sText               := 'ST053';
GVL_XTS.StationParameter[nStationParameter].rPosWait            :=   4100.0; // absolute modulo position
GVL_XTS.StationParameter[nStationParameter].rPosStop[1]         :=    270.0; // relative to rPosWait
GVL_XTS.StationParameter[nStationParameter].rPosStop[2]         :=    315.0; // relative to rPosWait
GVL_XTS.StationParameter[nStationParameter].rReleaseDistance    :=     10.0; // relative to Mover.ActPos
GVL_XTS.StationParameter[nStationParameter].rVelo               :=   2500.0;
GVL_XTS.StationParameter[nStationParameter].nConfiguredStopCount:= 2;

//---------------------------------------------------------------------------------------
//---------------------------------------------------------------------------------------
nStationParameter                    := 22;
GVL_XTS.StationParameter[nStationParameter].eType               := E_STATION_TYPE.STATION_PROCESS;
GVL_XTS.StationParameter[nStationParameter].sText               := 'ST061';
GVL_XTS.StationParameter[nStationParameter].rPosWait            :=   4750.0; // absolute modulo position
GVL_XTS.StationParameter[nStationParameter].rPosStop[1]         :=     90.0; // relative to rPosWait
GVL_XTS.StationParameter[nStationParameter].rReleaseDistance    :=     70.0; // relative to Mover.ActPos
GVL_XTS.StationParameter[nStationParameter].rVelo               :=   2500.0;

nStationParameter                    := 23;
GVL_XTS.StationParameter[nStationParameter].eType               := E_STATION_TYPE.STATION_PROCESS;
GVL_XTS.StationParameter[nStationParameter].sText               := 'ST062';
GVL_XTS.StationParameter[nStationParameter].rPosWait            :=   4750.0; // absolute modulo position
GVL_XTS.StationParameter[nStationParameter].rPosStop[1]         :=    180.0; // relative to rPosWait
GVL_XTS.StationParameter[nStationParameter].rReleaseDistance    :=     45.0; // relative to Mover.ActPos
GVL_XTS.StationParameter[nStationParameter].rVelo               :=   2500.0;

nStationParameter                    := 24;
GVL_XTS.StationParameter[nStationParameter].eType               := E_STATION_TYPE.STATION_PROCESS;
GVL_XTS.StationParameter[nStationParameter].sText               := 'ST063';
GVL_XTS.StationParameter[nStationParameter].rPosWait            :=   4750.0; // absolute modulo position
GVL_XTS.StationParameter[nStationParameter].rPosStop[1]         :=    270.0; // relative to rPosWait
GVL_XTS.StationParameter[nStationParameter].rReleaseDistance    :=     25.0; // relative to Mover.ActPos
GVL_XTS.StationParameter[nStationParameter].rVelo               :=   2500.0;


nStationParameter                    := 25;
GVL_XTS.StationParameter[nStationParameter].eType               := E_STATION_TYPE.STATION_PROCESS;
GVL_XTS.StationParameter[nStationParameter].sText               := 'ST064';
GVL_XTS.StationParameter[nStationParameter].rPosWait            :=   4750.0; // absolute modulo position
GVL_XTS.StationParameter[nStationParameter].rPosStop[1]         :=    360.0; // relative to rPosWait
GVL_XTS.StationParameter[nStationParameter].rReleaseDistance    :=     10.0; // relative to Mover.ActPos
GVL_XTS.StationParameter[nStationParameter].rVelo               :=   2500.0;

//---------------------------------------------------------------------------------------
//---------------------------------------------------------------------------------------
nStationParameter                    := 26;
GVL_XTS.StationParameter[nStationParameter].eType               := E_STATION_TYPE.STATION_PROCESS;
GVL_XTS.StationParameter[nStationParameter].sText               := 'ST071';
GVL_XTS.StationParameter[nStationParameter].rPosWait            :=   5600.0; // absolute modulo position
GVL_XTS.StationParameter[nStationParameter].rPosStop[1]         :=      0.0; // relative to rPosWait
GVL_XTS.StationParameter[nStationParameter].rReleaseDistance    :=    110.0; // relative to Mover.ActPos
GVL_XTS.StationParameter[nStationParameter].rVelo               :=   2500.0;

nStationParameter                    := 27;
GVL_XTS.StationParameter[nStationParameter].eType               := E_STATION_TYPE.STATION_PROCESS;
GVL_XTS.StationParameter[nStationParameter].sText               := 'ST072';
GVL_XTS.StationParameter[nStationParameter].rPosWait            :=   5700.0; // absolute modulo position
GVL_XTS.StationParameter[nStationParameter].rPosStop[1]         :=      0.0; // relative to rPosWait
GVL_XTS.StationParameter[nStationParameter].rReleaseDistance    :=     70.0; // relative to Mover.ActPos
GVL_XTS.StationParameter[nStationParameter].rVelo               :=   2500.0;

nStationParameter                    := 28;
GVL_XTS.StationParameter[nStationParameter].eType               := E_STATION_TYPE.STATION_PROCESS;
GVL_XTS.StationParameter[nStationParameter].sText               := 'ST073';
GVL_XTS.StationParameter[nStationParameter].rPosWait            :=   5800.0; // absolute modulo position
GVL_XTS.StationParameter[nStationParameter].rPosStop[1]         :=      0.0; // relative to rPosWait
GVL_XTS.StationParameter[nStationParameter].rReleaseDistance    :=     45.0; // relative to Mover.ActPos
GVL_XTS.StationParameter[nStationParameter].rVelo               :=   2500.0;

nStationParameter                    := 29;
GVL_XTS.StationParameter[nStationParameter].eType               := E_STATION_TYPE.STATION_PROCESS;
GVL_XTS.StationParameter[nStationParameter].sText               := 'ST074';
GVL_XTS.StationParameter[nStationParameter].rPosWait            :=   5900.0; // absolute modulo position
GVL_XTS.StationParameter[nStationParameter].rPosStop[1]         :=      0.0; // relative to rPosWait
GVL_XTS.StationParameter[nStationParameter].rReleaseDistance    :=     25.0; // relative to Mover.ActPos
GVL_XTS.StationParameter[nStationParameter].rVelo               :=   2500.0;

nStationParameter                    := 30;
GVL_XTS.StationParameter[nStationParameter].eType               := E_STATION_TYPE.STATION_PROCESS;
GVL_XTS.StationParameter[nStationParameter].sText               := 'ST075';
GVL_XTS.StationParameter[nStationParameter].rPosWait            :=   6000.0; // absolute modulo position
GVL_XTS.StationParameter[nStationParameter].rPosStop[1]         :=      0.0; // relative to rPosWait
GVL_XTS.StationParameter[nStationParameter].rReleaseDistance    :=     10.0; // relative to Mover.ActPos
GVL_XTS.StationParameter[nStationParameter].rVelo               :=   2500.0;

//---------------------------------------------------------------------------------------
//---------------------------------------------------------------------------------------
nStationParameter                    := 31;
GVL_XTS.StationParameter[nStationParameter].eType               := E_STATION_TYPE.STATION_PROCESS;
GVL_XTS.StationParameter[nStationParameter].sText               := 'ST081';
GVL_XTS.StationParameter[nStationParameter].rPosWait            :=   6900.0; // absolute modulo position
GVL_XTS.StationParameter[nStationParameter].rPosStop[1]         :=      0.0; // relative to rPosWait
GVL_XTS.StationParameter[nStationParameter].rReleaseDistance    :=    500.0; // relative to Mover.ActPos
GVL_XTS.StationParameter[nStationParameter].rVelo               :=   2500.0;

nStationParameter                    := 32;
GVL_XTS.StationParameter[nStationParameter].eType               := E_STATION_TYPE.STATION_PROCESS;
GVL_XTS.StationParameter[nStationParameter].sText               := 'ST082';
GVL_XTS.StationParameter[nStationParameter].rPosWait            :=   7000.0; // absolute modulo position
GVL_XTS.StationParameter[nStationParameter].rPosStop[1]         :=      0.0; // relative to rPosWait
GVL_XTS.StationParameter[nStationParameter].rReleaseDistance    :=    400.0; // relative to Mover.ActPos
GVL_XTS.StationParameter[nStationParameter].rVelo               :=   2500.0;

nStationParameter                    := 33;
GVL_XTS.StationParameter[nStationParameter].eType               := E_STATION_TYPE.STATION_PROCESS;
GVL_XTS.StationParameter[nStationParameter].sText               := 'ST083';
GVL_XTS.StationParameter[nStationParameter].rPosWait            :=   7100.0; // absolute modulo position
GVL_XTS.StationParameter[nStationParameter].rPosStop[1]         :=      0.0; // relative to rPosWait
GVL_XTS.StationParameter[nStationParameter].rReleaseDistance    :=    300.0; // relative to Mover.ActPos
GVL_XTS.StationParameter[nStationParameter].rVelo               :=   2500.0;

nStationParameter                    := 34;
GVL_XTS.StationParameter[nStationParameter].eType               := E_STATION_TYPE.STATION_PROCESS;
GVL_XTS.StationParameter[nStationParameter].sText               := 'ST084';
GVL_XTS.StationParameter[nStationParameter].rPosWait            :=   7200.0; // absolute modulo position
GVL_XTS.StationParameter[nStationParameter].rPosStop[1]         :=      0.0; // relative to rPosWait
GVL_XTS.StationParameter[nStationParameter].rReleaseDistance    :=    200.0; // relative to Mover.ActPos
GVL_XTS.StationParameter[nStationParameter].rVelo               :=   2500.0;

nStationParameter                    := 35;
GVL_XTS.StationParameter[nStationParameter].eType               := E_STATION_TYPE.STATION_PROCESS;
GVL_XTS.StationParameter[nStationParameter].sText               := 'ST085';
GVL_XTS.StationParameter[nStationParameter].rPosWait            :=   7300.0; // absolute modulo position
GVL_XTS.StationParameter[nStationParameter].rPosStop[1]         :=      0.0; // relative to rPosWait
GVL_XTS.StationParameter[nStationParameter].rReleaseDistance    :=    100.0; // relative to Mover.ActPos
GVL_XTS.StationParameter[nStationParameter].rVelo               :=   2500.0;

nStationParameter                    := 36;
GVL_XTS.StationParameter[nStationParameter].eType               := E_STATION_TYPE.STATION_PROCESS;
GVL_XTS.StationParameter[nStationParameter].sText               := 'ST086';
GVL_XTS.StationParameter[nStationParameter].rPosWait            :=   7400.0; // absolute modulo position
GVL_XTS.StationParameter[nStationParameter].rPosStop[1]         :=      0.0; // relative to rPosWait
GVL_XTS.StationParameter[nStationParameter].rReleaseDistance    :=     10.0; // relative to Mover.ActPos
GVL_XTS.StationParameter[nStationParameter].rVelo               :=   2500.0;

//---------------------------------------------------------------------------------------
//---------------------------------------------------------------------------------------
nStationParameter                    := 37;
GVL_XTS.StationParameter[nStationParameter].eType               := E_STATION_TYPE.STATION_PROCESS;
GVL_XTS.StationParameter[nStationParameter].sText               := 'START';
GVL_XTS.StationParameter[nStationParameter].rPosWait            :=   7800.0; // absolute modulo position
GVL_XTS.StationParameter[nStationParameter].rPosStop[1]         :=      0.0; // relative to rPosWait
GVL_XTS.StationParameter[nStationParameter].rReleaseDistance    :=     10.0; // relative to Mover.ActPos
GVL_XTS.StationParameter[nStationParameter].rVelo               :=   2500.0;

END_FUNCTION

// ---- _MSG/class/fb_MessageDataCtrl.TcPOU
FUNCTION_BLOCK fb_MessageDataCtrl EXTENDS fb_MessageData
VAR
  _stCtrl       : REFERENCE TO ST_MESSAGE_CTRL;
  _stState      : REFERENCE TO ST_MESSAGE_STATE;

  _eCmd,
  _eCmdOld      : E_MESSAGE_CTRL;

  _eResult,
  _eJobResult   : E_PROGRESS;

  _eState       : E_MESSAGE_STATE;

END_VAR

//-----------------------------------------------------------------------------
// check pointers
//-----------------------------------------------------------------------------
IF NOT Check()
THEN
  _eResult                      := E_PROGRESS.PROGRESS_ERROR;
  RETURN;
END_IF
//-----------------------------------------------------------------------------
// check date
// new message file for a new day
//-----------------------------------------------------------------------------
IF (FolderDate(_dtLocalTime) <> _sFolderDate)
THEN
  _bFileCreated                 := FALSE;
END_IF
//-----------------------------------------------------------------------------
//----------------------------------------------------------------------------- 
// copy to local for debug
_eCmd                         := _stCtrl.Cmd;

// cyclic check for command change
// get state for cmd
IF (_eCmd <> _eCmdOld)
THEN
  // get matching sdtate for Ctrl.Cmd
  _eState                     := Cmd(_eCmd);
  _eCmdOld                    := _eCmd;
END_IF


CASE _eResult
OF
  E_PROGRESS.PROGRESS_INVALID:
    _stState.State            := E_MESSAGE_STATE.MSG_STATE_NULL;

  E_PROGRESS.PROGRESS_ERROR:
    _stState.State            := _eState + E_PROGRESS.PROGRESS_ERROR;

  E_PROGRESS.PROGRESS_DONE:
    _stState.State            := _eState + E_PROGRESS.PROGRESS_DONE;

ELSE
  // work in progress
  // update progress for extern use
  _stState.State              := _eState + _eResult;

  CASE _eState
  OF
    E_MESSAGE_STATE.MSG_STATE_INIT:
      _eResult                := BuildFolder(TRUE);


    E_MESSAGE_STATE.MSG_STATE_IDLE:
      IF (_nMsgIndex < GVL_MSG_XTS.MAX_MESSAGE - GVL_MSG_XTS.MAX_MESSAGE/10)
      THEN
        _eResult              := E_PROGRESS.PROGRESS_WORKING;
      ELSE
        _eResult              := E_PROGRESS.PROGRESS_DONE;
        _nMsgIndex            := 0;
        // copy from attached list to local
        memcpy(ADR(_aWriteList), _pMsgList, SIZEOF(_aWriteList));
        // clear attached list
        memset(_pMsgList, 0, SIZEOF(_aWriteList));
      END_IF


    E_MESSAGE_STATE.MSG_STATE_WRITE:
      _eResult                := BuildFileData(TRUE);

  ELSE
      _eResult               := E_PROGRESS.PROGRESS_INVALID;
  END_CASE
END_CASE

METHOD BuildFileData : e_progress
VAR_INPUT
  Execute     : BOOL;
END_VAR
VAR_INST
  _nErrorId   : UDINT;
  _eState,
  _eRes       : E_PROGRESS;
  _eFlow      : E_MESSAGE_FLOW;

  _nStringLength  : UINT;
END_VAR
//-----------------------------------------------------------------------------
IF NOT Execute 
THEN
  _eRes                           := WriteData(FALSE);
  _eRes                           := BuildFolder(FALSE);
	_eState                         := E_PROGRESS.PROGRESS_INIT; 
END_IF 
//-----------------------------------------------------------------------------
IF NOT Check() 
THEN 
	BuildFileData                   := E_PROGRESS.PROGRESS_ERROR; 
	RETURN; 
END_IF
//-----------------------------------------------------------------------------
//-----------------------------------------------------------------------------
CASE _eState
OF
  E_PROGRESS.PROGRESS_INIT:
    IF Execute
    THEN
      _nErrorId                   := 0;
      _iStart 	                  := 1;
      _iEnd 		                  := SEL((_nMsgIndex > GVL_MSG_XTS.MAX_MESSAGE-1),
                                          _nMsgIndex,
                                          GVL_MSG_XTS.MAX_MESSAGE);

      memset(ADR(_sWriteData),0,SIZEOF(_sWriteData));

      IF (_sFolderDate <> FolderDate(_dtLocalTime))
      THEN
        _eState                   := E_PROGRESS.PROGRESS_PREPARE;
      ELSE
        _eState                   := E_PROGRESS.PROGRESS_BUSY;
        _eFlow                    := E_MESSAGE_FLOW.MSG_FLOW_LINE_START;
      END_IF
    END_IF
END_CASE
//-----------------------------------------------------------------------------
//-----------------------------------------------------------------------------
CASE _eState
OF
  E_PROGRESS.PROGRESS_PREPARE:
    _eRes                         := BuildFolder(TRUE);
    CASE _eRes
    OF
      E_PROGRESS.PROGRESS_DONE:
      _eState                     := E_PROGRESS.PROGRESS_BUSY;
      _eFlow                      := E_MESSAGE_FLOW.MSG_FLOW_LINE_START;

      E_PROGRESS.PROGRESS_ERROR:
      _eState                     := E_PROGRESS.PROGRESS_ERROR;
    END_CASE
END_CASE
//-----------------------------------------------------------------------------
//-----------------------------------------------------------------------------
CASE _eState
OF
  E_PROGRESS.PROGRESS_BUSY:
  CASE _eFlow
  OF
    E_MESSAGE_FLOW.MSG_FLOW_LINE_START:
      _eRes                       := BuildFolder(FALSE);
      _nErrIndex                  := 0; // rise and shine, all quarrels erased but not forgotten
      _nMsgIndex                  := 0;
  
      // copy from attached list to local
      memcpy(ADR(_aWriteList), _pMsgList, SIZEOF(_aWriteList));
  
      // clear attached list
      memset(_pMsgList, 0, SIZEOF(_aWriteList));


      _eFlow                      := E_MESSAGE_FLOW.MSG_FLOW_LINE_BUILD;
      _iCount                     := _iStart;
  END_CASE
  CASE _eFlow
  OF
    E_MESSAGE_FLOW.MSG_FLOW_LINE_BUILD:
      _eFlow                      := E_MESSAGE_FLOW.MSG_FLOW_LINE_CHECK;
      IF (_aWriteList[_iCount].eType > E_MessageType.eMessageEmpty)
      THEN
        _sTmp                     := TO_STRING(_aWriteList[_iCount].eType);
        _sTmp                     := Tc2_Standard.CONCAT(_sTmp, _sTab);
        _sTmp                     := Tc2_Standard.CONCAT(_sTmp, _aWriteList[_iCount].tTime);
        _sTmp                     := Tc2_Standard.CONCAT(_sTmp, _sTab);
        _sTmp                     := Tc2_Standard.CONCAT(_sTmp, Device_To_String(_aWriteList[_iCount].eDevice));
        _sTmp                     := Tc2_Standard.CONCAT(_sTmp, _sTab);
        _sTmp                     := Tc2_Standard.CONCAT(_sTmp, TO_STRING(_aWriteList[_iCount].eSubdevice));
        _sTmp                     := Tc2_Standard.CONCAT(_sTmp, _sTab);
        _sTmp                     := Tc2_Standard.CONCAT(_sTmp, TO_STRING(_aWriteList[_iCount].iErrorNumber));
        _sTmp                     := Tc2_Standard.CONCAT(_sTmp, _sTab);
        _sTmp                     := Tc2_Standard.CONCAT(_sTmp, _aWriteList[_iCount].sText);
        _sTmp                     := Tc2_Standard.CONCAT(_sTmp, _sNewLine);
        Builder(ADR(_sTmp), ADR(_sWriteData), StringLen(ADR(_sTmp)));
      END_IF
      _iCount                     := _iCount + 1;
  END_CASE
  CASE _eFlow
  OF
    E_MESSAGE_FLOW.MSG_FLOW_LINE_CHECK:
    IF NOT (_iCount > _iEnd)
    THEN
      _eFlow                      := E_MESSAGE_FLOW.MSG_FLOW_LINE_BUILD;
    ELSE
      _eState                     := E_PROGRESS.PROGRESS_WORKING;
      _eFlow                      := E_MESSAGE_FLOW.MSG_FLOW_WRITE_FILE_BUSY;
    END_IF
  END_CASE
END_CASE
//-----------------------------------------------------------------------------
//-----------------------------------------------------------------------------
CASE _eState
OF
  E_PROGRESS.PROGRESS_WORKING:
  CASE _eFlow
  OF
    E_MESSAGE_FLOW.MSG_FLOW_WRITE_FILE_BUSY:
      _nStringLength              := StringLen(ADR(_sWriteData));
      IF NOT (_nStringLength > 1)
      THEN
        _eState                   := E_PROGRESS.PROGRESS_DONE; 
       _eFlow                     := E_MESSAGE_FLOW.MSG_FLOW_WRITE_FILE_DONE;
      ELSE
        _eFlow                    := E_MESSAGE_FLOW.MSG_FLOW_WRITE_FILE_END;
        _eRes                     := WriteData(FALSE);
      END_IF
  END_CASE
  CASE _eFlow
  OF
    E_MESSAGE_FLOW.MSG_FLOW_WRITE_FILE_END:
      _eRes                       := WriteData(TRUE);

      IF (_eRes = E_PROGRESS.PROGRESS_ERROR)
      THEN
        _eState                   := E_PROGRESS.PROGRESS_ERROR;

      ELSIF (_eRes = E_PROGRESS.PROGRESS_DONE)
      THEN
        _eState                   := E_PROGRESS.PROGRESS_DONE;
        _eFlow                    := E_MESSAGE_FLOW.MSG_FLOW_WRITE_FILE_DONE;
        _eRes                     := WriteData(FALSE);
      END_IF
  END_CASE
END_CASE
//-----------------------------------------------------------------------------
//-----------------------------------------------------------------------------

BuildFileData                     := _eState;
END_METHOD

METHOD BuildFolder : e_progress
VAR_INPUT
  Execute           : BOOL;
END_VAR
VAR_INST
  _nErrorId   : UDINT;
  _eState     : E_PROGRESS;
  _eFlow      : E_MESSAGE_FLOW;
END_VAR
//-----------------------------------------------------------------------------
IF NOT Execute 
THEN 
	_eState                       := E_PROGRESS.PROGRESS_INIT; 
END_IF 
//-----------------------------------------------------------------------------
IF NOT Check() 
THEN 
	BuildFolder                   := E_PROGRESS.PROGRESS_ERROR; 
	RETURN; 
END_IF
//-----------------------------------------------------------------------------
//-----------------------------------------------------------------------------
CASE _eState
OF
  E_PROGRESS.PROGRESS_INIT:
    IF Execute
    THEN
      _nErrorId                 := 0;
      _bFileCreated             := FALSE;

      _sFolderDate              := FolderDate(_dtLocalTime);
      _eState                   := E_PROGRESS.PROGRESS_BUSY;
      _eFlow                    := E_MESSAGE_FLOW.MSG_FLOW_ROOT;
    END_IF
END_CASE
//-----------------------------------------------------------------------------
//-----------------------------------------------------------------------------
CASE _eState
OF
  E_PROGRESS.PROGRESS_BUSY:
  CASE _eFlow
  OF
    E_MESSAGE_FLOW.MSG_FLOW_ROOT:
      _eFlow                    := E_MESSAGE_FLOW.MSG_FLOW_ROOT_CREATE;
      _fbCreateDir.sPathName    := left(_pDirRoot^,len(_pDirRoot^)-1);
      _fbCreateDir(
              bExecute	        := FALSE);
    
    E_MESSAGE_FLOW.MSG_FLOW_ROOT_CREATE:
      (* create root folder *)
      _fbCreateDir(
              bExecute	        := TRUE);
      IF _fbCreateDir.bBusy
      THEN
        _eFlow                  := E_MESSAGE_FLOW.MSG_FLOW_ROOT_CREATE_BUSY;
      END_IF
    
    E_MESSAGE_FLOW.MSG_FLOW_ROOT_CREATE_BUSY:
      _fbCreateDir(
              bExecute	        := TRUE);
      IF NOT _fbCreateDir.bBusy
      THEN
        _eState                 := E_PROGRESS.PROGRESS_PREPARE;
        _eFlow                  := E_MESSAGE_FLOW.MSG_FLOW_FOLDER;
      END_IF
  END_CASE
END_CASE
//-----------------------------------------------------------------------------
//-----------------------------------------------------------------------------
CASE _eState
OF
  E_PROGRESS.PROGRESS_PREPARE:
  CASE _eFlow
  OF
    E_MESSAGE_FLOW.MSG_FLOW_FOLDER:
      _eFlow                    := E_MESSAGE_FLOW.MSG_FLOW_FOLDER_CREATE;
      _sFolderDate              := FolderDate(_dtLocalTime);
      _fbCreateDir.sPathName    := concat(_pDirRoot^, _sFolderDate);
      _fbCreateDir(
              bExecute	        := FALSE);
  
    E_MESSAGE_FLOW.MSG_FLOW_FOLDER_CREATE:
      (* create active folder *)
      _fbCreateDir(
              bExecute	        := TRUE);
      IF _fbCreateDir.bBusy
      THEN
        _eFlow                  := E_MESSAGE_FLOW.MSG_FLOW_FOLDER_CREATE_BUSY;
      END_IF
    
    E_MESSAGE_FLOW.MSG_FLOW_FOLDER_CREATE_BUSY:
      _fbCreateDir(
              bExecute	        := TRUE);
      IF NOT _fbCreateDir.bBusy
      THEN
        _eState                 := E_PROGRESS.PROGRESS_CHECK;
        _eFlow                  := E_MESSAGE_FLOW.MSG_FLOW_FILE_CREATE_DONE;
        _fbCreateDir(
                bExecute	      := FALSE);
      END_IF
  END_CASE
END_CASE
//-----------------------------------------------------------------------------
//-----------------------------------------------------------------------------
CASE _eState
OF
  E_PROGRESS.PROGRESS_CHECK:
  CASE _eFlow
  OF
    E_MESSAGE_FLOW.MSG_FLOW_FILE_CREATE_DONE:
      _eState                   := E_PROGRESS.PROGRESS_DONE;
      _bFileCreated             := TRUE;

      // build complete file path
      _sTmp                     := concat(concat(_pFileRoot^, _sFolderDate),'.txt');
      _sTmp                     := concat('\', _sTmp);
      _sFilename                := concat(_fbCreateDir.sPathName, _sTmp);
  END_CASE
END_CASE

BuildFolder                     := _eState;
END_METHOD

METHOD Check : BOOL
VAR_INPUT
END_VAR

IF NOT __ISVALIDREF(_stCtrl)
THEN
  _eCheck       := E_MESSAGE_CHECK.POINTER_CTRL_INVALID;
  RETURN;
END_IF

IF NOT __ISVALIDREF(_stState)
THEN
  _eCheck       := E_MESSAGE_CHECK.POINTER_STATE_INVALID;
  RETURN;
END_IF
//-----------------------------------------------------------------
//-----------------------------------------------------------------
IF NOT (_dtLocalTime <> 0)
THEN
  _eCheck       := E_MESSAGE_CHECK.POINTER_TIME_INVALID;
  RETURN;
END_IF

IF NOT (_pMsgList <> 0)
THEN
  _eCheck       := E_MESSAGE_CHECK.POINTER_LIST_INVALID;
  RETURN;
END_IF

IF NOT (_pFileRoot <> 0)
THEN
  _eCheck       := E_MESSAGE_CHECK.POINTER_ROOT_FILE_INVALID;
  RETURN;
END_IF

IF NOT (_pDirRoot <> 0)
THEN
  _eCheck       := E_MESSAGE_CHECK.POINTER_ROOT_DIR_INVALID;
  RETURN;
END_IF

IF NOT __ISVALIDREF(_nMsgIndex)
THEN
  _eCheck       := E_MESSAGE_CHECK.POINTER_MSG_IDX_INVALID;
  RETURN;
END_IF

IF NOT __ISVALIDREF(_nErrIndex)
THEN
  _eCheck       := E_MESSAGE_CHECK.POINTER_ERR_IDX_INVALID;
  RETURN;
END_IF


_eCheck         := E_MESSAGE_CHECK.CHECK_DONE;
Check           := TRUE;
END_METHOD

METHOD Cmd : e_message_state
VAR_INPUT
  Command     : e_message_ctrl;
END_VAR


CASE Command
OF
  E_MESSAGE_CTRL.MSG_CTRL_NULL:
    _eResult                    := E_PROGRESS.PROGRESS_INVALID;
    Cmd                         := E_MESSAGE_STATE.MSG_STATE_NULL;

  E_MESSAGE_CTRL.MSG_CTRL_INIT:
    _eResult                    := BuildFolder(FALSE);
    Cmd                         := E_MESSAGE_STATE.MSG_STATE_INIT;

  E_MESSAGE_CTRL.MSG_CTRL_IDLE:
    _eResult                    := BuildFileData(FALSE);
    Cmd                         := E_MESSAGE_STATE.MSG_STATE_IDLE;

  E_MESSAGE_CTRL.MSG_CTRL_WRITE:
    _eResult                    := BuildFileData(FALSE);
    Cmd                         := E_MESSAGE_STATE.MSG_STATE_WRITE;
    IF (_nMsgIndex = 0)
    THEN
       // go back to sleep
      _eResult                := E_PROGRESS.PROGRESS_DONE;
    END_IF
ELSE
    //_eResult                    := E_PROGRESS.PROGRESS_ERROR;
    Cmd                         := E_MESSAGE_STATE.MSG_STATE_NULL;
END_CASE
END_METHOD

PROPERTY Ctrl : REFERENCE to ST_MESSAGE_CTRL
SET
_stCtrl ref= Ctrl;
END_SET
END_PROPERTY

PROPERTY FileCreated : bool
GET
FileCreated := _bFileCreated;
END_GET
END_PROPERTY

PROPERTY State : REFERENCE TO ST_MESSAGE_STATE
SET
_stState ref= State;
END_SET
END_PROPERTY

END_FUNCTION_BLOCK

// ---- _XML/types/fb_XmlRead.TcPOU
FUNCTION_BLOCK fb_XmlRead
VAR_INPUT
  bExecute      : BOOL;
  sFilePath     : STRING(255);(*File and Path Name*)
  sXPath        : STRING;     (*Dataentry in XML file*)
  pData         : pvoid;      (*pointer to Datafield*)
  diSize        : UDINT;      (*size of datafield*)
END_VAR
VAR_OUTPUT
  bBusy         : BOOL;
  bDone         : BOOL;
  bError        : BOOL;
  nError        : UDINT;
END_VAR
VAR
  rtrigIn       : Tc2_Standard.R_TRIG;
  ftrigIn       : Tc2_Standard.F_TRIG;
  diStep        : DINT;
  sMsg          : ARRAY[1..10] OF STRING;
  iMsg          : DINT := 1;

  fbReadData    : Tc2_XmlDataSrv.FB_XmlSrvRead;
END_VAR


rtrigIn(CLK:= bExecute);
ftrigIn(CLK:= bExecute);

IF rtrigIn.Q
THEN
  bBusy := TRUE;
  bDone := FALSE;
  bError:= FALSE;
  diStep  := 10;
END_IF

IF ftrigIn.Q
THEN
  fbReadData(bExecute := FALSE);
  bBusy := FALSE;
  bDone := FALSE;
  bError:= FALSE;
  diStep  := 0;
END_IF


CASE diStep OF

  10:
    sMsg[iMsg] := 'start: ';
    iMsg := iMsg + 1;
    fbReadData(bExecute := FALSE);
    diStep := 15;

  15:
    fbReadData(
      bExecute := TRUE,
      sNetId:= '', 
      ePath       := PATH_GENERIC, 
      nMode       := XMLSRV_SKIPMISSING, 
      pSymAddr    := pData, 
      cbSymSize   := diSize, 
      sFilePath   := sFilePath, 
      sXPath      := sXPath, 
      bExecute:= , 
      tTimeout    := T#5S, 
      bBusy=> , 
      bError=> , 
      nErrId=> nError);

    IF fbReadData.bBusy
    THEN
      sMsg[iMsg] := 'busy: ';
      iMsg := iMsg + 1;
      diStep := 20;
    END_IF

  20:
    fbReadData();
    IF NOT fbReadData.bError
    THEN
      nError := 0;
      IF NOT fbReadData.bBusy
      THEN
        sMsg[iMsg] := 'done: ';
        iMsg := iMsg + 1;
        fbReadData(bExecute := FALSE);
        diStep := 30;
      END_IF
    ELSE
      nError := fbReadData.nErrId;
      sMsg[iMsg] := 'error: ';
      sMsg[iMsg] := concat(sMsg[iMsg], TO_STRING(fbReadData.nErrId));
      iMsg := iMsg + 1;
      diStep := 99;
    END_IF

  30:
    bBusy := FALSE;
    bDone := TRUE;

  99:
    bBusy := FALSE;
    bError:= TRUE;
END_CASE

IF (iMsg > 10) THEN iMsg :=1; END_IF

END_FUNCTION_BLOCK

// ---- _XML/types/fb_XmlWrite.TcPOU
FUNCTION_BLOCK fb_XmlWrite
VAR_INPUT
  bExecute      : BOOL;
  sFilePath     : STRING(255);(*File and Path Name*)
  sXPath        : STRING;     (*Dataentry in XML file*)
  pData         : pvoid;      (*pointer to Datafield*)
  diSize        : UDINT;      (*size of datafield*)
END_VAR
VAR_OUTPUT
  bBusy         : BOOL;
  bDone         : BOOL;
  bError        : BOOL;
  nError        : UDINT;
END_VAR
VAR
  rtrigIn       : Tc2_Standard.R_TRIG;
  ftrigIn       : Tc2_Standard.F_TRIG;
  diStep        : DINT;
  sMsg          : ARRAY[1..10] OF STRING;
  iMsg          : DINT := 1;

  fbWriteData   : Tc2_XmlDataSrv.FB_XmlSrvWrite;
END_VAR


rtrigIn(CLK:= bExecute);
ftrigIn(CLK:= bExecute);


IF rtrigIn.Q
THEN
  bBusy := TRUE;
  bDone := FALSE;
  bError:= FALSE;
  diStep  := 10;
END_IF

IF ftrigIn.Q
THEN
  fbWriteData(bExecute := FALSE);
  diStep  := 0;
END_IF

CASE diStep OF

  0:
    bBusy := FALSE;
    bDone := FALSE;
    bError:= FALSE;

  10:
    sMsg[iMsg] := 'start: ';
    iMsg := iMsg + 1;
    fbWriteData(bExecute := FALSE);
    diStep := 15;

  15:
    fbWriteData(
      bExecute := TRUE,
      sNetId:= '', 
      ePath       := PATH_GENERIC, 
      nMode       := Tc2_XmlDataSrv.XMLSRV_ADDMISSING, 
      pSymAddr    := pData, 
      cbSymSize   := diSize, 
      sFilePath   := sFilePath, 
      sXPath      := sXPath, 
      bExecute:= , 
      tTimeout    := T#5S, 
      bBusy=> , 
      bError=> , 
      nErrId=> );

    IF fbWriteData.bBusy
    THEN
      sMsg[iMsg] := 'busy: ';
      iMsg := iMsg + 1;
      diStep := 20;
    END_IF

  20:
    fbWriteData();
    IF NOT fbWriteData.bError
    THEN
      nError := 0;
      IF NOT fbWriteData.bBusy
      THEN
        sMsg[iMsg] := 'done: ';
        iMsg := iMsg + 1;
        fbWriteData(bExecute := FALSE);
        diStep := 30;
      END_IF
    ELSE
      IF fbWriteData.nErrId <> 0
      THEN
        nError := fbWriteData.nErrId;
        sMsg[iMsg] := 'error: ';
        sMsg[iMsg] := concat(sMsg[iMsg], TO_STRING(fbWriteData.nErrId));
        iMsg := iMsg + 1;

        fbWriteData(bExecute := FALSE);
        diStep := 99;
      END_IF
    END_IF

  30:
    bBusy := FALSE;
    bDone := TRUE;

  99:
    bBusy  := FALSE;
    bError := TRUE;
END_CASE

IF (iMsg > 10) THEN iMsg :=1; END_IF

END_FUNCTION_BLOCK

// ---- XTS_TRANSPORT/_Visualization/GROUP_VISU.TcVIS
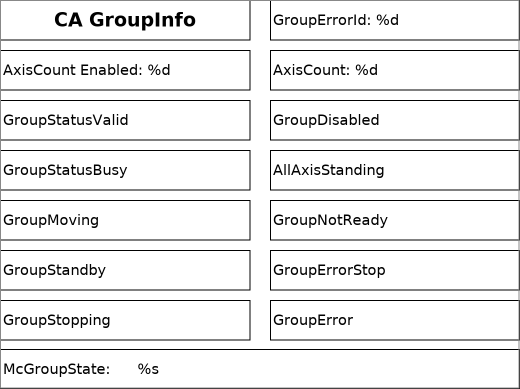
VISUALIZATION GROUP_VISU  // 520x389
VAR_IN_OUT
	stGroupInfo   : ST_GROUP_INFO;
  sGroupState   : string(60);
END_VAR
    Rectangle (0,100 250x40), "GroupStatusValid", colour toggle: stGroupInfo.GroupStatusValid
    Rectangle (0,150 250x40), "GroupStatusBusy", colour toggle: stGroupInfo.GroupStatusBusy
    Rectangle (0,200 250x40), "GroupMoving", colour toggle: stGroupInfo.GroupMoving
    Rectangle (270,250 250x40), "GroupErrorStop", colour toggle: stGroupInfo.GroupErrorStop
    Rectangle (270,200 250x40), "GroupNotReady", colour toggle: stGroupInfo.GroupNotReady
    Rectangle (0,250 250x40), "GroupStandby", colour toggle: stGroupInfo.GroupStandby
    Rectangle (0,300 250x40), "GroupStopping", colour toggle: stGroupInfo.GroupStopping
    Rectangle (270,100 250x40), "GroupDisabled", colour toggle: stGroupInfo.GroupDisabled
    Rectangle (270,150 250x40), "AllAxisStanding", colour toggle: stGroupInfo.AllAxesStanding
    Rectangle (270,300 250x40), "GroupError", colour toggle: stGroupInfo.GroupError
    Rectangle (270,0 250x40), "GroupErrorId: %d", text variable: stGroupInfo.GroupErrorId
    Rectangle (270,50 250x40), "AxisCount: %d", text variable: stGroupInfo.AxisCount
    Rectangle (0,349 520x40), "McGroupState: %s", text variable: sGroupState
    Rectangle (0,0 250x40), "CA GroupInfo"
    Rectangle (0,50 250x40), "AxisCount Enabled: %d", text variable: stGroupInfo.AxisCountEnabled
END_VISUALIZATION

// ---- XTS_TRANSPORT/_Visualization/MOVER_VISU.TcVIS
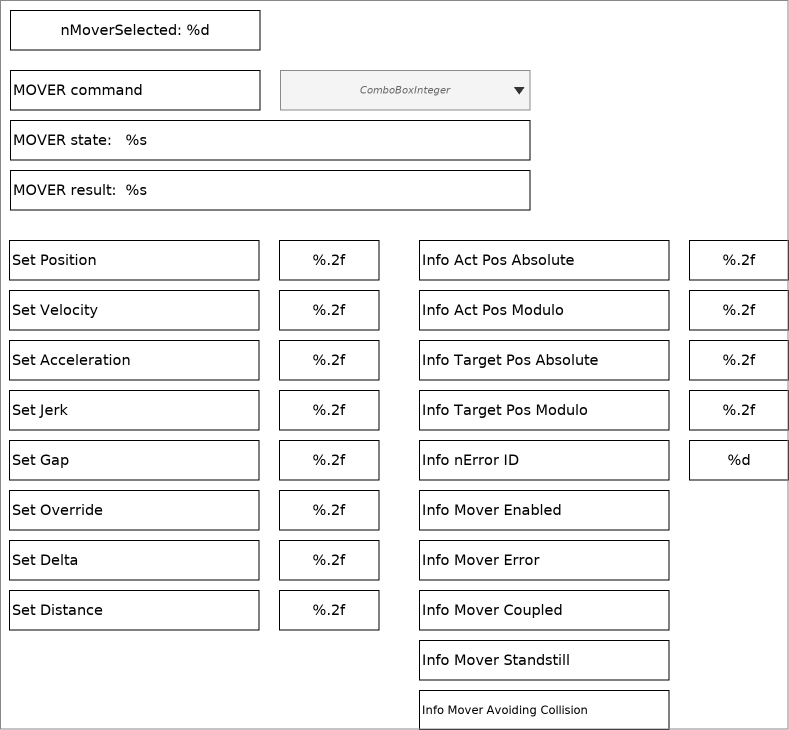
VISUALIZATION MOVER_VISU  // 789x730
    Rectangle (10,10 250x40), "nMoverSelected: %d", text variable: MAIN.nMoverSelected
        OnMouseClick: write the text variable via VisuDialogs.Numpad, min 1, max MAX_MOVER, title 'Selected Mover'
    Rectangle (10,120 520x40), "MOVER state: %s", text variable: MAIN.sMoverState
    Rectangle (10,70 250x40), "MOVER command"
    ComboBoxInteger (280,70 250x40), variable: GVL_XTS.MoverCtrl[MAIN.nMoverSelected].Cmd, text list: 'TL_E_CTRL_MOVER'
    Rectangle (10,170 520x40), "MOVER result: %s", text variable: MAIN.sMoverResult
    Rectangle (9,240 250x40), "Set Position"
    Rectangle (9,290 250x40), "Set Velocity"
    Rectangle (9,340 250x40), "Set Acceleration"
    Rectangle (9,390 250x40), "Set Jerk"
    Rectangle (9,440 250x40), "Set Gap"
    Rectangle (9,490 250x40), "Set Override"
    Rectangle (9,540 250x40), "Set Delta"
    Rectangle (9,590 250x40), "Set Distance"
    Rectangle (279,240 100x40), "%.2f", text variable: GVL_XTS.MoveData[MAIN.nMoverSelected].rPos
        OnMouseClick: write the text variable via Default
    Rectangle (279,290 100x40), "%.2f", text variable: GVL_XTS.MoveData[MAIN.nMoverSelected].rVelo
        OnMouseClick: write the text variable via Default
    Rectangle (279,340 100x40), "%.2f", text variable: GVL_XTS.MoveData[MAIN.nMoverSelected].rAcc
        OnMouseClick: write the text variable via Default
    Rectangle (279,390 100x40), "%.2f", text variable: GVL_XTS.MoveData[MAIN.nMoverSelected].rJerk
        OnMouseClick: write the text variable via Default
    Rectangle (279,440 100x40), "%.2f", text variable: GVL_XTS.MoveData[MAIN.nMoverSelected].rGap
        OnMouseClick: write the text variable via Default
    Rectangle (279,490 100x40), "%.2f", text variable: GVL_XTS.MoveData[MAIN.nMoverSelected].rOverride
        OnMouseClick: write the text variable via Default
    Rectangle (279,540 100x40), "%.2f", text variable: GVL_XTS.MoveData[MAIN.nMoverSelected].rDelta
        OnMouseClick: write the text variable via Default
    Rectangle (279,590 100x40), "%.2f", text variable: GVL_XTS.MoveData[MAIN.nMoverSelected].rDistance
        OnMouseClick: write the text variable via Default
    Rectangle (419,240 250x40), "Info Act Pos Absolute"
    Rectangle (419,290 250x40), "Info Act Pos Modulo"
    Rectangle (419,340 250x40), "Info Target Pos Absolute"
    Rectangle (419,390 250x40), "Info Target Pos Modulo"
    Rectangle (419,440 250x40), "Info nError ID"
    Rectangle (689,240 100x40), "%.2f", text variable: GVL_XTS.MoverInfo[MAIN.nMoverSelected].rAbsActPos
    Rectangle (689,290 100x40), "%.2f", text variable: GVL_XTS.MoverInfo[MAIN.nMoverSelected].rModuloActPos
    Rectangle (689,340 100x40), "%.2f", text variable: GVL_XTS.MoverInfo[MAIN.nMoverSelected].rAbsTargetPos
    Rectangle (689,390 100x40), "%.2f", text variable: GVL_XTS.MoverInfo[MAIN.nMoverSelected].rModuloTargetPos
    Rectangle (689,440 100x40), "%d", text variable: GVL_XTS.MoverInfo[MAIN.nMoverSelected].nErrorId
    Rectangle (419,490 250x40), "Info Mover Enabled", colour toggle: GVL_XTS.MoverInfo[MAIN.nMoverSelected].bMoverEnabled
    Rectangle (419,540 250x40), "Info Mover Error", colour toggle: GVL_XTS.MoverInfo[MAIN.nMoverSelected].bMoverError
    Rectangle (419,590 250x40), "Info Mover Coupled", colour toggle: GVL_XTS.MoverInfo[MAIN.nMoverSelected].bMoverCoupled
    Rectangle (419,640 250x40), "Info Mover Standstill", colour toggle: GVL_XTS.MoverInfo[MAIN.nMoverSelected].bMoverStandstill
    Rectangle (419,690 250x40), "Info Mover Avoiding Collision", colour toggle: GVL_XTS.MoverInfo[MAIN.nMoverSelected].bMoverAvoidingCollision
END_VISUALIZATION

// ---- XTS_TRANSPORT/_Visualization/SELECTOR_VISU.TcVIS
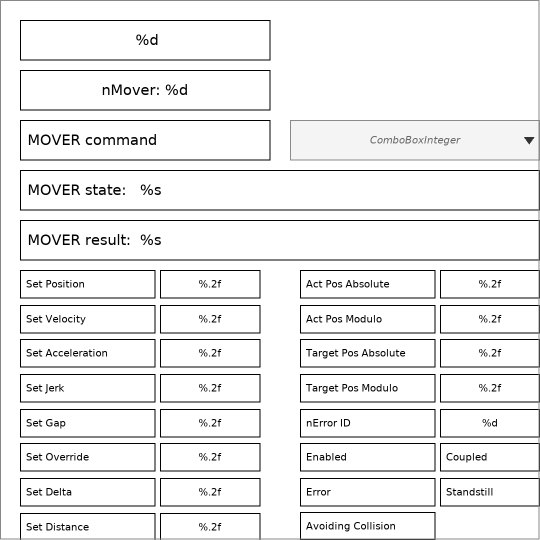
VISUALIZATION SELECTOR_VISU  // 540x540
    Frame (10,10 530x530)
        shows T_MOVER_SELECTOR(Control := GVL_XTS.SelectorCtrl, State := GVL_XTS.SelectorState, sState := MAIN.sSelectorState, sResult := MAIN.sSelectorResult)
END_VISUALIZATION

// ---- XTS_TRANSPORT/_Visualization/STATION_VISU.TcVIS
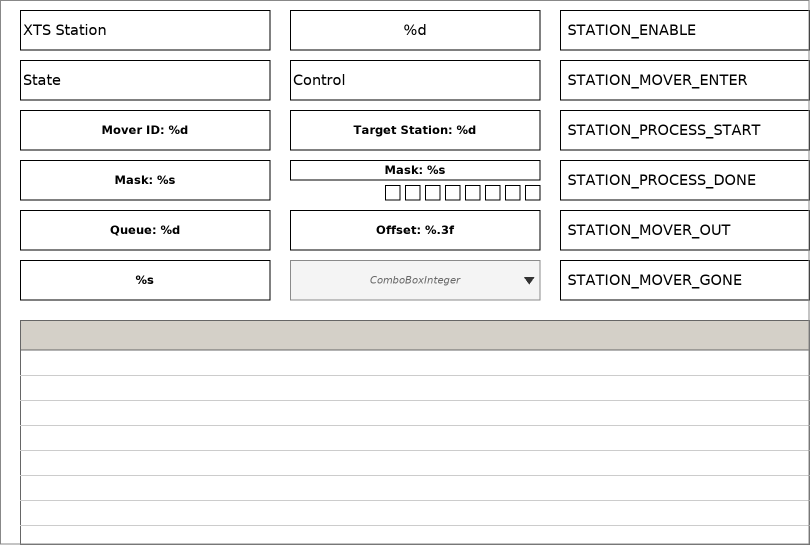
VISUALIZATION STATION_VISU  // 810x545
    Rectangle (20,10 250x40), "XTS Station"
    Rectangle (290,10 250x40), "%d", text variable: MAIN_XTS.nStationSelected
        OnMouseClick: write the text variable via VisuDialogs.Numpad, min 1, max MAX_STATION, title 'Selected Station'
    Rectangle (20,60 250x40), "State"
    Rectangle (290,60 250x40), "Control"
    Rectangle (20,210 250x40), "Queue: %d", text variable: GVL_XTS.StationState[MAIN_XTS.nStationSelected].nQueue
    Rectangle (20,110 250x40), "Mover ID: %d", text variable: GVL_XTS.StationState[MAIN_XTS.nStationSelected].nMoverId
    Rectangle (20,160 250x40), "Mask: %s", text variable: MAIN_XTS.sStationStateMask
    Rectangle (20,260 250x40), "%s", text variable: MAIN_XTS.sStationState
    ComboBoxInteger (290,260 250x40), variable: GVL_XTS.StationCtrl[MAIN_XTS.nStationSelected].eCmd, text list: 'TL_E_CTRL_STATION'
    Rectangle (290,210 250x40), "Offset: %.3f", text variable: GVL_XTS.StationCtrl[MAIN_XTS.nStationSelected].rOffset
    Rectangle (290,110 250x40), "Target Station: %d", text variable: GVL_XTS.StationCtrl[MAIN_XTS.nStationSelected].nTargetStation
        OnMouseClick: write the text variable via VisuDialogs.Numpad, min 1, max MAX_STATION, title 'Target Station'
    Rectangle (290,160 250x20), "Mask: %s", text variable: MAIN_XTS.sStationCtrlMask
    Rectangle (525,185 15x15)
        toggle GVL_XTS.StationCtrl[MAIN_XTS.nStationSelected].nMask.0
    Rectangle (505,185 15x15)
        toggle GVL_XTS.StationCtrl[MAIN_XTS.nStationSelected].nMask.1
    Rectangle (485,185 15x15)
        toggle GVL_XTS.StationCtrl[MAIN_XTS.nStationSelected].nMask.2
    Rectangle (465,185 15x15)
        toggle GVL_XTS.StationCtrl[MAIN_XTS.nStationSelected].nMask.3
    Rectangle (445,185 15x15)
        toggle GVL_XTS.StationCtrl[MAIN_XTS.nStationSelected].nMask.4
    Rectangle (425,185 15x15)
        toggle GVL_XTS.StationCtrl[MAIN_XTS.nStationSelected].nMask.5
    Rectangle (405,185 15x15)
        toggle GVL_XTS.StationCtrl[MAIN_XTS.nStationSelected].nMask.6
    Rectangle (385,185 15x15)
        toggle GVL_XTS.StationCtrl[MAIN_XTS.nStationSelected].nMask.7
    Rectangle (560,10 250x40), "STATION_ENABLE", colour toggle: MAIN_XTS.bStationEnable
        OnMouseClick: execute { GVL_XTS.StationCtrl[MAIN_XTS.nStationSelected].Cmd := E_STATION_CTRL.STATION_ENABLE; }
    Rectangle (560,60 250x40), "STATION_MOVER_ENTER", colour toggle: MAIN_XTS.bStationEnter
        OnMouseClick: execute { GVL_XTS.StationCtrl[MAIN_XTS.nStationSelected].Cmd := E_STATION_CTRL.STATION_MOVER_ENTER; }
    Rectangle (560,110 250x40), "STATION_PROCESS_START", colour toggle: MAIN_XTS.bStationStart
        OnMouseClick: execute { GVL_XTS.StationCtrl[MAIN_XTS.nStationSelected].Cmd := E_STATION_CTRL.STATION_PROCESS_START; }
    Rectangle (560,160 250x40), "STATION_PROCESS_DONE", colour toggle: MAIN_XTS.bStationDone
        OnMouseClick: execute { GVL_XTS.StationCtrl[MAIN_XTS.nStationSelected].Cmd := E_STATION_CTRL.STATION_PROCESS_DONE; }
    Rectangle (560,210 250x40), "STATION_MOVER_OUT", colour toggle: MAIN_XTS.bStationOut
        OnMouseClick: execute { GVL_XTS.StationCtrl[MAIN_XTS.nStationSelected].Cmd := E_STATION_CTRL.STATION_MOVER_OUT; }
    Rectangle (560,260 250x40), "STATION_MOVER_GONE", colour toggle: MAIN_XTS.bStationGone
        OnMouseClick: execute { GVL_XTS.StationCtrl[MAIN_XTS.nStationSelected].Cmd := E_STATION_CTRL.STATION_MOVER_GONE; }
    Table (20,320 790x225), data array: MAIN_XTS.tStationSelectedQueue
        p3854506369: MAIN_XTS.tStationSelectedQueue[INDEX].nMoverId
        p1892666644: MAIN_XTS.tStationSelectedQueue[INDEX].nTargetStation
        p338671338: MAIN_XTS.tStationSelectedQueue[INDEX].nMask
        p2170511999: MAIN_XTS.tStationSelectedQueue[INDEX].rOffset
        p1014161805: GVL_XTS_CONSTANTS.MAX_LIST_NODES - 1 + INT#1
END_VISUALIZATION

// ---- XTS_TRANSPORT/_Visualization/textlists/TL_E_CTRL_MOVER.TcTLO
TEXTLIST TL_E_CTRL_MOVER
  0 = 'MOVER_NULL'
  1 = 'MOVER_ENABLE'
  2 = 'MOVER_DISABLE'
  4 = 'MOVER_MOVE_TO_POS_CA'
  5 = 'MOVER_SEND_TO_POS_CA'
  6 = 'MOVER_HALT'
  7 = 'MOVER_GEAR_IN'
  8 = 'MOVER_GEAR_IN_POS_CA'
  9 = 'MOVER_GEAR_OUT'
  10 = 'MOVER_RESET'
  3 = 'MOVER_MOVE_TO_POS'
   = ''
END_TEXTLIST

// ---- XTS_TRANSPORT/_Visualization/textlists/TL_E_CTRL_STATION.TcTLO
TEXTLIST TL_E_CTRL_STATION
  0 = 'STATION_CTRL_NULL'
  1 = 'STATION_INIT'
  10 = 'STATION_DISABLE'
  11 = 'STATION_ENABLE'
  20 = 'STATION_MOVER_ENTER'
  21 = 'STATION_MOVER_ENTER_RETRY'
  22 = 'STATION_MOVER_SEND'
  30 = 'STATION_PROCESS_START'
  31 = 'STATION_PROCESS_DONE'
  50 = 'STATION_MOVER_OUT'
  51 = 'STATION_MOVER_OUT_RETRY'
  60 = 'STATION_MOVER_GONE'
   = ''
END_TEXTLIST

// ---- XTS_TRANSPORT/_Visualization/textlists/TL_E_CTRL_TRANSPORT.TcTLO
TEXTLIST TL_E_CTRL_TRANSPORT
  0 = 'CMD_NULL'
  10 = 'CMD_INIT'
  11 = 'CMD_IDLE'
  20 = 'CMD_MOVER_ENABLE'
  21 = 'CMD_MOVER_DISABLE'
  22 = 'CMD_MOVER_HALT_CA'
  23 = 'CMD_MOVER_STOP'
  30 = 'CMD_GROUP_CLEAR'
  31 = 'CMD_GROUP_BUILD'
  32 = 'CMD_GROUP_ENABLE'
  33 = 'CMD_GROUP_STOP'
  40 = 'CMD_TRANSPORT_START'
  41 = 'CMD_TRANSPORT_RESTART'
   = ''
END_TEXTLIST

// ---- XTS_TRANSPORT/_Visualization/textlists/TL_E_CTRL_XPU.TcTLO
TEXTLIST TL_E_CTRL_XPU
  0 = 'XTS_CMD_NULL'
  10 = 'XTS_CMD_INIT'
  30 = 'XTS_IDLE'
   = ''
END_TEXTLIST

// ---- XTS_TRANSPORT/_Visualization/types/T_MOVER_SELECTOR.TcVIS
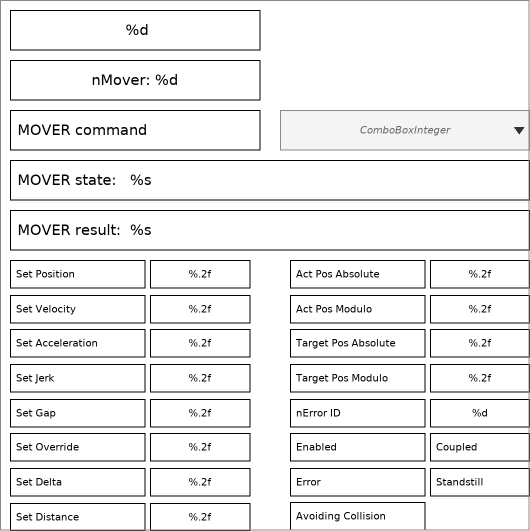
VISUALIZATION T_MOVER_SELECTOR  // 530x531
VAR_IN_OUT
	Control     : ST_MOVER_SELECTOR_CTRL;
  State       : ST_MOVER_SELECTOR_STATE;
  sState      : STRING;
  sResult     : STRING;
END_VAR
    Rectangle (10,60 250x40), "nMover: %d", text variable: Control.Mover
        OnMouseClick: write the text variable via VisuDialogs.Numpad, min 1, max MAX_MOVER, title 'Selected Mover'
    Rectangle (10,10 250x40), "%d", text variable: Control.Selector, text list: 'TL_E_MOVER_SELECTOR'
        OnMouseClick: write the text variable via VisuDialogs.Numpad, min 1, max MAX_MOVER, title 'Selected Mover'
    Rectangle (10,160 520x40), "MOVER state: %s", text variable: sState
    Rectangle (10,110 250x40), "MOVER command"
    ComboBoxInteger (280,110 250x40), variable: Control.Control.Cmd, text list: 'TL_E_CTRL_MOVER'
    Rectangle (10,210 520x40), "MOVER result: %s", text variable: sResult
    Rectangle (10,260 135x28), "Set Position"
    Rectangle (10,295 135x28), "Set Velocity"
    Rectangle (10,329 135x28), "Set Acceleration"
    Rectangle (10,364 135x28), "Set Jerk"
    Rectangle (10,399 135x28), "Set Gap"
    Rectangle (10,433 135x28), "Set Override"
    Rectangle (10,468 135x28), "Set Delta"
    Rectangle (10,503 135x28), "Set Distance"
    Rectangle (150,260 100x28), "%.2f", text variable: Control.Data.rPos
        OnMouseClick: write the text variable via Default
    Rectangle (150,295 100x28), "%.2f", text variable: Control.Data.rVelo
        OnMouseClick: write the text variable via Default
    Rectangle (150,329 100x28), "%.2f", text variable: Control.Data.rAcc
        OnMouseClick: write the text variable via Default
    Rectangle (150,364 100x28), "%.2f", text variable: Control.Data.rJerk
        OnMouseClick: write the text variable via Default
    Rectangle (150,399 100x28), "%.2f", text variable: Control.Data.rGap
        OnMouseClick: write the text variable via Default
    Rectangle (150,433 100x28), "%.2f", text variable: Control.Data.rOverride
        OnMouseClick: write the text variable via Default
    Rectangle (150,468 100x28), "%.2f", text variable: Control.Data.rDelta
        OnMouseClick: write the text variable via Default
    Rectangle (150,503 100x28), "%.2f", text variable: Control.Data.rDistance
        OnMouseClick: write the text variable via Default
    Rectangle (290,260 135x28), "Act Pos Absolute"
    Rectangle (290,295 135x28), "Act Pos Modulo"
    Rectangle (290,329 135x28), "Target Pos Absolute"
    Rectangle (290,364 135x28), "Target Pos Modulo"
    Rectangle (290,399 135x28), "nError ID"
    Rectangle (430,260 100x28), "%.2f", text variable: GVL_XTS.MoverInfo[MAIN.nMoverSelected].rAbsActPos
    Rectangle (430,295 100x28), "%.2f", text variable: GVL_XTS.MoverInfo[MAIN.nMoverSelected].rModuloActPos
    Rectangle (430,329 100x28), "%.2f", text variable: GVL_XTS.MoverInfo[MAIN.nMoverSelected].rAbsTargetPos
    Rectangle (430,364 100x28), "%.2f", text variable: GVL_XTS.MoverInfo[MAIN.nMoverSelected].rModuloTargetPos
    Rectangle (430,399 100x28), "%d", text variable: GVL_XTS.MoverInfo[MAIN.nMoverSelected].nErrorId
    Rectangle (290,433 135x28), "Enabled", colour toggle: GVL_XTS.MoverInfo[MAIN.nMoverSelected].bMoverEnabled
    Rectangle (290,468 135x28), "Error", colour toggle: GVL_XTS.MoverInfo[MAIN.nMoverSelected].bMoverError
    Rectangle (430,433 100x28), "Coupled", colour toggle: GVL_XTS.MoverInfo[MAIN.nMoverSelected].bMoverCoupled
    Rectangle (430,468 100x28), "Standstill", colour toggle: GVL_XTS.MoverInfo[MAIN.nMoverSelected].bMoverStandstill
    Rectangle (290,502 135x28), "Avoiding Collision", colour toggle: GVL_XTS.MoverInfo[MAIN.nMoverSelected].bMoverAvoidingCollision
END_VISUALIZATION

// ---- XTS_TRANSPORT/_Visualization/XPU_VISU.TcVIS
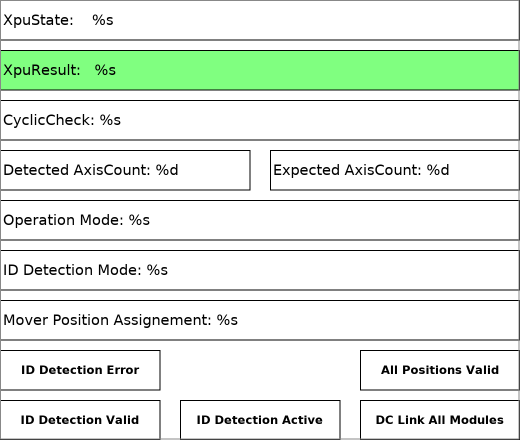
VISUALIZATION XPU_VISU  // 520x440
VAR_IN_OUT
	stXpuState    : ST_XPU_STATE;
  stXpuInfo     : ST_XPU_INFO;
  stXpuStrings  : ST_XPU_STRINGS;
END_VAR
    Rectangle (0,100 520x40), "CyclicCheck: %s", text variable: stXpuStrings.sXpuCyclicCheck
    Rectangle (0,0 520x40), "XpuState: %s", text variable: stXpuStrings.sXpuState
    Rectangle (0,50 520x40), "XpuResult: %s", text variable: stXpuStrings.sXpuResult, colour toggle: (MAIN.eXpuResult = E_PROGRESS.PROGRESS_ERROR)
    Rectangle (360,350 160x40), "All Positions Valid", colour toggle: stXpuInfo.AllPositionsValid
    Rectangle (0,350 160x40), "ID Detection Error", colour toggle: stXpuInfo.IdDetectionError
    Rectangle (0,400 160x40), "ID Detection Valid", colour toggle: stXpuInfo.IdDetectionValid
    Rectangle (180,400 160x40), "ID Detection Active", colour toggle: stXpuInfo.IdDetectionActive
    Rectangle (0,200 520x40), "Operation Mode: %s", text variable: stXpuStrings.sXpuOpMode
    Rectangle (0,250 520x40), "ID Detection Mode: %s", text variable: stXpuStrings.sXpuMoverId_DetectionMode
    Rectangle (0,300 520x40), "Mover Position Assignement: %s", text variable: stXpuStrings.sXpuMoverPosAssignement
    Rectangle (270,150 250x40), "Expected AxisCount: %d", text variable: stXpuInfo.nExpectedAxisCount
    Rectangle (0,150 250x40), "Detected AxisCount: %d", text variable: stXpuInfo.nDetectedAxisCount
    Rectangle (360,400 160x40), "DC Link All Modules", colour toggle: stXpuState.DcLink
END_VISUALIZATION

// ---- XTS_TRANSPORT/_Visualization/XTS_TRANSPORT.TcVIS
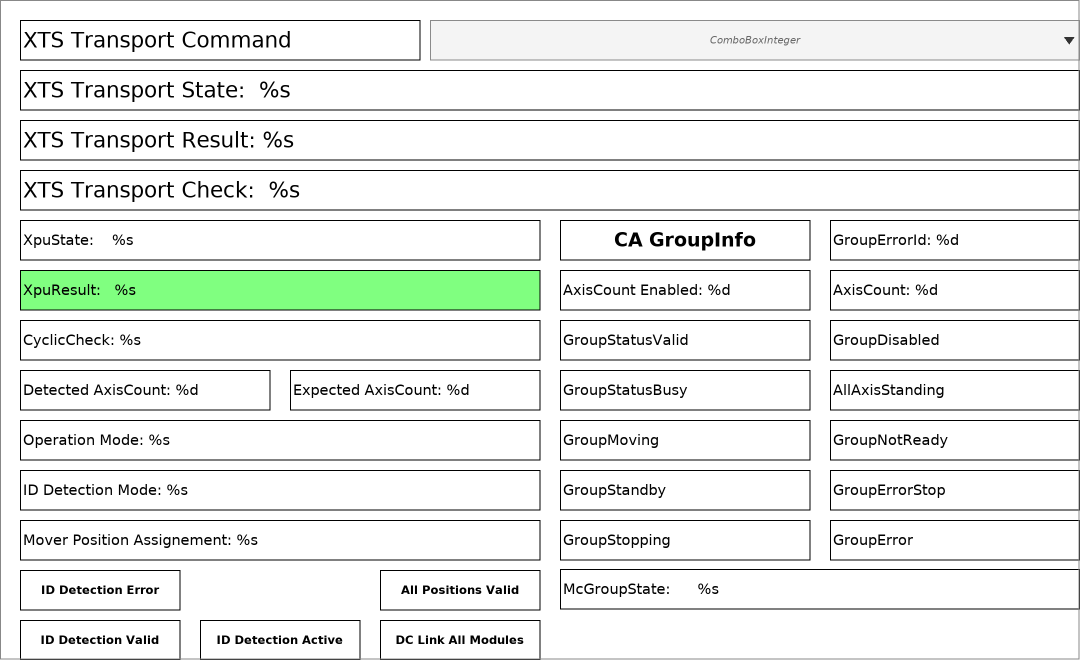
VISUALIZATION XTS_TRANSPORT  // 1080x660
    Rectangle (20,20 400x40), "XTS Transport Command"
    ComboBoxInteger (430,20 650x40), variable: GVL_XTS.XtsTransportCtrl.Cmd, text list: 'TL_E_CTRL_TRANSPORT'
    Rectangle (20,70 1060x40), "XTS Transport State: %s", text variable: MAIN_XTS.sTransportState
    Rectangle (20,120 1060x40), "XTS Transport Result: %s", text variable: MAIN_XTS.sTransportResult
    Rectangle (20,170 1060x40), "XTS Transport Check: %s", text variable: MAIN_XTS.sTransportCheck
    Frame (20,220 520x440)
        shows XPU_VISU(stXpuState := GVL_XTS.XtsTransportState.XpuState, stXpuInfo := GVL_XTS.XtsTransportState.XpuInfo, stXpuStrings := MAIN_XTS.stXpuStrings)
    Frame (560,220 520x390)
        shows GROUP_VISU(stGroupInfo := GVL_XTS.XtsTransportState.GroupInfo, sGroupState := MAIN_XTS.sCaGroupState)
END_VISUALIZATION

// ---- _MSG/types/TL_E_MESSAGETYPE.TcTLO
TEXTLIST TL_E_MESSAGETYPE
  0 = 'eMessageEmpty'
  1 = 'eMessageError'
  2 = 'eMessageWarning'
  3 = 'eMessageInfo'
  4 = 'eMessageVerbose'
   = ''
END_TEXTLIST
